No03: NOP   0;
NoXX: NOP   0;
NETWORK
TITLE =ASW_6030: Active step germinating
//      U     "MAL1S024Par".Par.FlagProcess.ProcessActive;
//      SPBN  tuen;
//
//// copy stepnr
//      L     "MAL1S024Par".Par.ParIntMachine.ActualStep;
//      T     "MAL1S024Par".Par.ParIntProcess.ActualStep;
//// set step conditions
//
//// Case where process is starting during loading
//      U     "MAL1S024Par".Par.FlagProcess.ProcessActive;
//      UN    "MAL1S024Par".Par.FlagFunction_1.StepLoading; // Step loading
//      SPBN  e003;
//// lifting devices must be in highest position
//      L       WinCoS_BIW01_09PLC1BIW01_02.Ma.Par.ParPositionTopRightUnits;
////Malting Plant OAO Belsolod Ivanonvo Weissrussland
//      L     50; // 50mm offset
//      +I    ;
//      T     "MAL1S024Par".Par.MachineValue.SOLLWERT_HUBZUG1_HOEHE;
//      L       WinCoS_BIW01_09PLC1BIW01_02.Ma.Par.ParPositionTopLeftUnits;
////Malting Plant OAO Belsolod Ivanonvo Weissrussland
//      L     50; // 50mm offset
//      +I    ;
//      T     "MAL1S024Par".Par.MachineValue.SOLLWERT_HUBZUG2_HOEHE;
//      L     5;
//      T     WinCoS_BIW01_09PLC1BIW01_02.Ma.Par.ParTolPosition;
//e003: NOP   0;
//
//// reset turning cmds
//
//// save turning cmds from prev.step
//      L     "MAL1S024Par".Par.ParIntMachine.ActualStep;
//      L     "MAL1S024Par".Par.ParIntProcess.PrevStep1stTurn;
//      <>I   ;
//      SPB   sav1;
//      U     "MAL1S024Par".Par.FlagProcess2.Turning1WithSpraying;
//      =     "MAL1S024Par".Par.Switches1.StaOn08; // Turning1WithSpraying
//      U     "MAL1S024Par".Par.FlagProcess2.Turning1WithDosing;
//      =     "MAL1S024Par".Par.Switches1.StaOn09; // Turning1WithDosing
//sav1: NOP   0;
//      L     "MAL1S024Par".Par.ParIntMachine.ActualStep;
//      L     "MAL1S024Par".Par.ParIntProcess.PrevStep2ndTurn;
//      <>I   ;
//      SPB   sav2;
//      U     "MAL1S024Par".Par.FlagProcess2.Turning2WithSpraying;
//      =     "MAL1S024Par".Par.Switches1.StaOn10; // Turning2WithSpraying
//      U     "MAL1S024Par".Par.FlagProcess2.Turning2WithDosing;
//      =     "MAL1S024Par".Par.Switches1.StaOn11; // Turning2WithDosing
//sav2: NOP   0;
//
//      SET   ;
//      R     "MAL1S024Par".Par.FlagProcess2.Turning1WithoutSpraying;
//      R     "MAL1S024Par".Par.FlagProcess2.Turning1WithSpraying;
//      R     "MAL1S024Par".Par.FlagProcess2.Turning1WithDosing;
//      R     "MAL1S024Par".Par.FlagProcess2.Turning2WithoutSpraying;
//      R     "MAL1S024Par".Par.FlagProcess2.Turning2WithSpraying;
//      R     "MAL1S024Par".Par.FlagProcess2.Turning2WithDosing;
//
//// Delta Temp to switch to next step
//      L     "MAL1S024Par".StepAct.DeltaTempSwitchpointStep;
//      L     L#0;
//      >D   ;
//      =     "MAL1S024Par".Par.FlagProcess1.DeltaTempNextStep;
//// Max Temp to switch to next step
//      L     "MAL1S024Par".StepAct.MaxTempAboveFloorStep;
//      L     L#0;
//      >D   ;
//      =     "MAL1S024Par".Par.FlagProcess1.MaxTempNextStep;
//
//// position waste air see sub 6050
//
//// basic speed fan see sub 6040
//
//// air humifidication
//      L     1;
//      L     "MAL1S024Par".StepAct.AirMoisten;   // On/Off
//      ==I;  // air humifidication on
//      U     WinCoS_BIW01_09PLC1BIW01_02.Ma.StStartedFwd; //Malting Plant OAO
//Belsolod Ivanonvo Weissrussland
//      =     "MAL1S024Par".Par.FlagProcess.AirHumidificationValve1; // air
//humifidication valve 1 on
//      U(    ; // air humifidication on
//      L     "MAL1S024Par".Par.ParIntMachine.TargetSpeedGermFan; // germinating
//fan is running
//      L     40; // fanspeed > 40%
//      >I    ; // muss noch in Istwert getauscht werden JV
//      )     ; // fanspeed > 40%
//      =     "MAL1S024Par".Par.FlagProcess.AirHumidificationValve2;
//
//// air cooling
//      L     "MAL1S024Par".StepAct.Cooling;
//      L   1;  // Activate Cooling System = 1 (yes)
//      ==I;
//      =     "MAL1S024Par".Par.FlagProcess.Cooling; // request cooling
//
//      U     "MAL1S024Par".Par.FlagProcess.ProcessActive;
//      U     "MAL1S024".PCRead.Step.StReady;
//      UN    "MAL1S024Par".Par.FlagFunction_1.StepLoading;
//      SPBN  e630;
//
//// turning 1
//      UN    "MAL1S024Par".Par.FlagProcess2.StartSecondTurningRound; // Turn
//from PrevStep
//      U(;
//      L     "MAL1S024Par".StepAct.StartTurningRound_1;
//      L     0;
//      >=D;                  // negative, no turning 1
//      );
//      U(    ;
//      O(    ; // Nach Rezept
//      L     "MAL1S024Par".ActTimeStepProcess.StepTimeActHourTotal; // Steptime
//in hours overall
//      L     "MAL1S024Par".StepAct.StartTurningRound_1;
//      ==I   ;
//      UN     WinCoS_BIW01_09PLC1BIW01_02.Ma.StAdjusted; // target position
//turning reached
//      )     ;
//      O(    ; // Selbsthaltung
//      L     "MAL1S024Par".ActTimeStepProcess.StepTimeActHourTotal; // Steptime
//in hours overall
//      L     "MAL1S024Par".StepAct.StartTurningRound_1;
//      <>I   ;
//      U     "MAL1S024Par".Par.FlagProcess2.StartFirstTurningRound;
//      )     ;
//      )     ;
//      S     "MAL1S024Par".Par.FlagProcess2.Turning1WithoutSpraying;
//      S     "MAL1S024Par".Par.FlagFunction_1.TurningStart;
//// turning 1 with spraying
//      U(    ;
//      L     1;
//      L     "MAL1S024Par".StepAct.TurningWithSpraying_1;
//      ==I;    // turning 1 with spraying on
//      U(    ;
//      L     "MAL1S024Par".Par.ParIntMachine.ActualStep;
//      L     "MAL1S024Par".Par.ParIntProcess.PrevStep1stTurn;
//      ==I   ;
//      )     ;
//      )     ;
//      O(    ;
//      L     "MAL1S024Par".Par.ParIntMachine.ActualStep;
//      L     "MAL1S024Par".Par.ParIntProcess.PrevStep1stTurn;
//      <>I   ;
//      U     "MAL1S024Par".Par.Switches1.StaOn08; // Turning1WithSpraying
//      )     ;
//      U     "MAL1S024Par".Par.FlagProcess2.Turning1WithoutSpraying;
//      S     "MAL1S024Par".Par.FlagProcess2.Turning1WithSpraying;
//// turning 1 with spraying and GA3
//      U(    ;
//      L     1;
//      L     "MAL1S024Par".StepAct.TurningWithDosing_1;
//      ==I;    // turning 1 with spraying on
//      U(    ;
//      L     "MAL1S024Par".Par.ParIntMachine.ActualStep;
//      L     "MAL1S024Par".Par.ParIntProcess.PrevStep1stTurn;
//      ==I   ;
//      )     ;
//      )     ;
//      O(    ;
//      L     "MAL1S024Par".Par.ParIntMachine.ActualStep;
//      L     "MAL1S024Par".Par.ParIntProcess.PrevStep1stTurn;
//      <>I   ;
//      U     "MAL1S024Par".Par.Switches1.StaOn09; // Turning1WithDosing
//      )     ;
//      U     "MAL1S024Par".Par.FlagProcess2.Turning1WithoutSpraying;
//      S     "MAL1S024Par".Par.FlagProcess2.Turning1WithSpraying;
//      S     "MAL1S024Par".Par.FlagProcess2.Turning1WithDosing;
//
//      U     "MAL1S024Par".Par.FlagProcess2.Turning1WithoutSpraying;
//      U     "MAL1S024Par".Par.FlagFunction_1.TurningStart;
//      UN     WinCoS_BIW01_09PLC1BIW01_02.Ma.StAdjusted; // target position
//turning reached
//      FP    "MAL1S024Par".Par.FlagProcess2.StartFirstTurningFP;
//      S     "MAL1S024Par".Par.FlagProcess2.StartFirstTurningRound;
//
//      U     WinCoS_BIW01_09PLC1BIW01_02.Ma.StAdjusted; // target position
//turning reached
//      O(    ;
//      L     "MAL1S024Par".ActTimeStepProcess.StepTimeActHourTotal; // Steptime
//in hours overall
//      L     "MAL1S024Par".StepAct.StartTurningRound_1;
//      >I    ;
//      U     WinCoS_BIW01_09PLC1BIW01_02.Ma.StAdjusted; // target position
//turning reached
//      )     ;
//      U     "MAL1S024Par".Par.FlagProcess2.StartFirstTurningRound;
//      R     "MAL1S024Par".Par.FlagProcess2.StartFirstTurningRound;
//
//      U     "MAL1S024Par".Par.FlagProcess2.StartFirstTurningFP;
//      SPB   trn1;
//      L     "MAL1S024Par".Par.ParIntMachine.ActualStep;
//      T     "MAL1S024Par".Par.ParIntProcess.PrevStep1stTurn;
//trn1: NOP   0;
//
//// turning 2
//      UN    "MAL1S024Par".Par.FlagProcess2.StartFirstTurningRound; // Unsinngie
//Rezeptwerte
//      U(;
//      L     1;
//      L     "MAL1S024Par".StepAct.StartTurningRound_2;
//      ==I    ;
//      );
//      U(    ;
//      O(    ; // Nach Rezept
//      L     "MAL1S024Par".ActTimeStepProcess.StepTimeActHourTotal; // Steptime
//in hours overall
//      L     "MAL1S024Par".StepAct.StartTurningRound_2;
//      ==I   ;
//      UN     WinCoS_BIW01_09PLC1BIW01_02.Ma.StAdjusted; // target position
//turning reached
//      )     ;
//      O(    ; // Selbsthaltung
//      L     "MAL1S024Par".ActTimeStepProcess.StepTimeActHourTotal; // Steptime
//in hours overall
//      L     "MAL1S024Par".StepAct.StartTurningRound_2;
//      <>I   ;
//      U     "MAL1S024Par".Par.FlagProcess2.StartSecondTurningRound;
//      )     ;
//      )     ;
//      S     "MAL1S024Par".Par.FlagProcess2.Turning2WithoutSpraying;
//      S     "MAL1S024Par".Par.FlagFunction_1.TurningStart;
//// turning 2 with spraying
//      U(    ;
//      L     1;
//      L     "MAL1S024Par".StepAct.TurningWithSpraying_2;
//      ==I    ;
//      U(    ;
//      L     "MAL1S024Par".Par.ParIntMachine.ActualStep;
//      L     "MAL1S024Par".Par.ParIntProcess.PrevStep2ndTurn;
//      ==I   ;
//      )     ;
//      )     ;
//      O(    ;
//      L     "MAL1S024Par".Par.ParIntMachine.ActualStep;
//      L     "MAL1S024Par".Par.ParIntProcess.PrevStep2ndTurn;
//      <>I   ;
//      U     "MAL1S024Par".Par.Switches1.StaOn10; // Turning2WithSpraying
//      )     ;
//      U     "MAL1S024Par".Par.FlagProcess2.Turning2WithoutSpraying;
//      S     "MAL1S024Par".Par.FlagProcess2.Turning2WithSpraying;
//// turning 2 with spraying and GA3
//      U(    ;
//      L     1;
//      L     "MAL1S024Par".StepAct.TurningWithDosing_2;
//      ==I;    // turning 2 with spraying and GA3 on
//      U(    ;
//      L     "MAL1S024Par".Par.ParIntMachine.ActualStep;
//      L     "MAL1S024Par".Par.ParIntProcess.PrevStep2ndTurn;
//      ==I   ;
//      )     ;
//      )     ;
//      O(    ;
//      L     "MAL1S024Par".Par.ParIntMachine.ActualStep;
//      L     "MAL1S024Par".Par.ParIntProcess.PrevStep2ndTurn;
//      <>I   ;
//      U     "MAL1S024Par".Par.Switches1.StaOn11; // Turning2WithDosing
//      )     ;
//      U     "MAL1S024Par".Par.FlagProcess2.Turning2WithoutSpraying;
//      S     "MAL1S024Par".Par.FlagProcess2.Turning2WithSpraying;
//      S     "MAL1S024Par".Par.FlagProcess2.Turning2WithDosing;
//
//      U     "MAL1S024Par".Par.FlagProcess2.Turning2WithoutSpraying;
//      U     "MAL1S024Par".Par.FlagFunction_1.TurningStart;
//      UN     WinCoS_BIW01_09PLC1BIW01_02.Ma.StAdjusted; // target position
//turning reached
//      FP    "MAL1S024Par".Par.FlagProcess2.StartSecondTurningFP;
//      S     "MAL1S024Par".Par.FlagProcess2.StartSecondTurningRound;
//
//      U     WinCoS_BIW01_09PLC1BIW01_02.Ma.StAdjusted; // target position
//turning reached
//      O(    ;
//      L     "MAL1S024Par".ActTimeStepProcess.StepTimeActHourTotal; // Steptime
//in hours overall
//      L     "MAL1S024Par".StepAct.StartTurningRound_2;
//      >I    ;
//      U     WinCoS_BIW01_09PLC1BIW01_02.Ma.StAdjusted; // target position
//turning reached
//      )     ;
//      U     "MAL1S024Par".Par.FlagProcess2.StartSecondTurningRound;
//      R     "MAL1S024Par".Par.FlagProcess2.StartSecondTurningRound;
//
//      U     "MAL1S024Par".Par.FlagProcess2.StartSecondTurningFP;
//      SPB   trn2;
//      L     "MAL1S024Par".Par.ParIntMachine.ActualStep;
//      T     "MAL1S024Par".Par.ParIntProcess.PrevStep2ndTurn;
//trn2: NOP   0;
////Fix Speed for Turning
//      U     "MAL1S024Par".Par.FlagProcess2.Turning1WithoutSpraying;
//      O     "MAL1S024Par".Par.FlagProcess2.Turning1WithSpraying;
//      O     "MAL1S024Par".Par.FlagProcess2.Turning2WithoutSpraying;
//      O     "MAL1S024Par".Par.FlagProcess2.Turning2WithSpraying;
//      U    M 50.0;
//      SPBN  SpdT;
//      L     15; // 15Hz
//      T     "MAL1S024Par".Par.MachineValue.SollwertFahrantrieb;
//SpdT: NOP   0;
//
//// find turning direction
//      U     "MAL1S024Par".Par.FlagGen.TurningStarted;
//      O(    ;
//      UN    "MAL1S024Par".Par.FlagProcess2.Turning1WithoutSpraying;
//      UN    "MAL1S024Par".Par.FlagProcess2.Turning2WithoutSpraying;
//      )     ;
//      SPB   tuen;
//      L     "MAL1S024Par".Par.ParIntMachine.TargetPosTravDriTurnRigt; // 370° =
//endposition turning right
//      T     WinCoS_BIW01_09PLC1BIW01_02.Ma.InPositionTarget; // target position
//turning reached
//
//      U(    ;
//      L     WinCoS_BIW01_09PLC1BIW01_02.Ma.OutPositionAngle;
//      L     1800;
//      <I    ; // condition turning right (clockwise)
//      )     ;
//      S     "MAL1S024Par".Par.FlagFunction_1.TurningRight;
//      S     "MAL1S024Par".Par.FlagGen.TurningStarted;
//// - Correct effect of ILO Mode
//      L       WinCoS_BIW01_09PLC1BIW01_02.Ma.Par.ParPositionTopLeftUnits;
////Malting Plant OAO Belsolod Ivanonvo Weissrussland
//      T     "MAL1S024Par".Par.MachineValue.SOLLWERT_HUBZUG1_HOEHE;
//      L       WinCoS_BIW01_09PLC1BIW01_02.Ma.Par.ParPositionTopRightUnits;
////Malting Plant OAO Belsolod Ivanonvo Weissrussland
//      T     "MAL1S024Par".Par.MachineValue.SOLLWERT_HUBZUG2_HOEHE;
//      SPB   E603   ;
//      L     "MAL1S024Par".Par.ParIntMachine.TargetPosTravDriTurnLeft; // 0° =
//endposition turning left
//      T     WinCoS_BIW01_09PLC1BIW01_02.Ma.InPositionTarget; // target position
//turning reached
//
//      U(    ;
//      L     WinCoS_BIW01_09PLC1BIW01_02.Ma.OutPositionAngle;
//      L     1800;
//      >=I   ; // condition turning left (counterclockwise)
//      )     ;
//      S     "MAL1S024Par".Par.FlagFunction_1.TurningLeft;
//      S     "MAL1S024Par".Par.FlagGen.TurningStarted;
//// - Correct effect of ILO Mode
//      L       WinCoS_BIW01_09PLC1BIW01_02.Ma.Par.ParPositionTopLeftUnits;
////Malting Plant OAO Belsolod Ivanonvo Weissrussland
//      T     "MAL1S024Par".Par.MachineValue.SOLLWERT_HUBZUG1_HOEHE;
//      L       WinCoS_BIW01_09PLC1BIW01_02.Ma.Par.ParPositionTopRightUnits;
////Malting Plant OAO Belsolod Ivanonvo Weissrussland
//      T     "MAL1S024Par".Par.MachineValue.SOLLWERT_HUBZUG2_HOEHE;
//      SPB   E603   ;
//tuen: NOP   0;
//// - Case of fast speed to protect a 2nd start during same hours as finsihed
//      O(    ; // Nach Rezept
//      L     "MAL1S024Par".ActTimeStepProcess.StepTimeActHourTotal; // Steptime
//in hours overall
//      L     "MAL1S024Par".StepAct.StartTurningRound_1;
//      ==I   ;
//      U     WinCoS_BIW01_09PLC1BIW01_02.Ma.StAdjusted; // target position
//turning reached
//      U     "MAL1S024Par".Par.FlagFunction_1.TurningStart;
//      )     ;
//      O(    ; // Nach Rezept
//      L     "MAL1S024Par".ActTimeStepProcess.StepTimeActHourTotal; // Steptime
//in hours overall
//      L     "MAL1S024Par".StepAct.StartTurningRound_2;
//      ==I   ;
//      U     WinCoS_BIW01_09PLC1BIW01_02.Ma.StAdjusted; // target position
//turning reached
//      U     "MAL1S024Par".Par.FlagFunction_1.TurningStart;
//      )     ;
//      SPB   e603;
//
//// reset turning right (clockwise)
//      U     "MAL1S024Par".Par.FlagFunction_1.TurningRight;
//      U(    ;
//      O      WinCoS_BIW01_09PLC1BIW01_02.Ma.StAdjusted; // target position
//turning reached
//      O(    ;
//      L     WinCoS_BIW01_09PLC1BIW01_02.Ma.OutPositionAngle;
//      L     WinCoS_BIW01_09PLC1BIW01_02.Ma.Par.ParTolPosition;
//      +I    ;
//      L     "MAL1S024Par".Par.ParIntMachine.TargetPosTravDriTurnRigt;
//      >=I   ;
//      )     ;
//      )     ;
//      R     "MAL1S024Par".Par.FlagFunction_1.TurningRight;
//      R     "MAL1S024Par".Par.FlagFunction_1.TurningStart;
//
//// reset turning left (counterclockwise)
//      U     "MAL1S024Par".Par.FlagFunction_1.TurningLeft;
//      U(    ;
//      O     WinCoS_BIW01_09PLC1BIW01_02.Ma.StAdjusted; // target position
//turning reached
//      O(    ;
//      L     WinCoS_BIW01_09PLC1BIW01_02.Ma.OutPositionAngle;
//      L     WinCoS_BIW01_09PLC1BIW01_02.Ma.Par.ParTolPosition;
//      -I    ;
//      L     "MAL1S024Par".Par.ParIntMachine.TargetPosTravDriTurnLeft;
//      <=I   ;
//      )     ;
//      )     ;
//      R     "MAL1S024Par".Par.FlagFunction_1.TurningLeft;
//      R     "MAL1S024Par".Par.FlagFunction_1.TurningStart;
//
//// reset turning flag
//      U     "MAL1S024Par".Par.FlagGen.TurningStarted;
//      UN    "MAL1S024Par".Par.FlagProcess2.Turning1WithoutSpraying;
//      UN    "MAL1S024Par".Par.FlagProcess2.Turning2WithoutSpraying;
//      O(    ;
//      U     "MAL1S024Par".Par.FlagGen.TurningStarted;
//      U     WinCoS_BIW01_09PLC1BIW01_02.Ma.StAdjusted; // target position
//turning reached
//      )     ;
//      ON    "MAL1S024Par".Par.FlagProcess.ProcessActive;
//      R     "MAL1S024Par".Par.FlagGen.TurningStarted;
//      R     "MAL1S024Par".Par.FlagProcess2.Turning1WithoutSpraying;
//      R     "MAL1S024Par".Par.FlagProcess2.Turning2WithoutSpraying;
//      R     "MAL1S024Par".Par.FlagFunction_1.TurningStart;
//e630: NOP   0;
//      UN    "MAL1S024Par".Par.FlagProcess.ProcessActive;
//      R     "MAL1S024Par".Par.FlagProcess2.StartFirstTurningRound;
//      R     "MAL1S024Par".Par.FlagProcess2.StartSecondTurningRound;
//
//e603: NOP   0;
//E603: NOP   0;
      U     "MAL1S024Par".Par.FlagProcess.ProcessActive;
      SPBN  tuen;

// copy stepnr
      L     "MAL1S024Par".Par.ParIntMachine.ActualStep;
      T     "MAL1S024Par".Par.ParIntProcess.ActualStep;
// set step conditions

// reset turning cmds

// save turning cmds from prev.step
      L     "MAL1S024Par".Par.ParIntMachine.ActualStep;
      L     "MAL1S024Par".Par.ParIntProcess.PrevStep1stTurn;
      <>I   ;
      SPB   sav1;
      U     "MAL1S024Par".Par.FlagProcess2.Turning1WithSpraying;
      =     "MAL1S024Par".Par.Switches1.StaOn08; // Turning1WithSpraying
      U     "MAL1S024Par".Par.FlagProcess2.Turning1WithDosing;
      =     "MAL1S024Par".Par.Switches1.StaOn09; // Turning1WithDosing
sav1: NOP   0;
      L     "MAL1S024Par".Par.ParIntMachine.ActualStep;
      L     "MAL1S024Par".Par.ParIntProcess.PrevStep2ndTurn;
      <>I   ;
      SPB   sav2;
      U     "MAL1S024Par".Par.FlagProcess2.Turning2WithSpraying;
      =     "MAL1S024Par".Par.Switches1.StaOn10; // Turning2WithSpraying
      U     "MAL1S024Par".Par.FlagProcess2.Turning2WithDosing;
      =     "MAL1S024Par".Par.Switches1.StaOn11; // Turning2WithDosing
sav2: NOP   0;

      SET   ;
      R     "MAL1S024Par".Par.FlagProcess2.Turning1WithoutSpraying;
      R     "MAL1S024Par".Par.FlagProcess2.Turning1WithSpraying;
      R     "MAL1S024Par".Par.FlagProcess2.Turning1WithDosing;
      R     "MAL1S024Par".Par.FlagProcess2.Turning2WithoutSpraying;
      R     "MAL1S024Par".Par.FlagProcess2.Turning2WithSpraying;
      R     "MAL1S024Par".Par.FlagProcess2.Turning2WithDosing;

// Delta Temp to switch to next step
      L     "MAL1S024Par".StepAct.DeltaTempSwitchpointStep;
      L     L#0;
      >D    ;
      =     "MAL1S024Par".Par.FlagProcess1.DeltaTempNextStep;
// Max Temp to switch to next step
      L     "MAL1S024Par".StepAct.MaxTempAboveFloorStep;
      L     L#0;
      >D    ;
      =     "MAL1S024Par".Par.FlagProcess1.MaxTempNextStep;

// position waste air see sub 6050

// basic speed fan see sub 6040

// air humifidication

// air cooling
      L     "MAL1S024Par".StepAct.Cooling;
      L     1; // Activate Cooling System = 1 (yes)
      ==I   ;
      =     "MAL1S024Par".Par.FlagProcess.Cooling; // request cooling

      U     "MAL1S024Par".Par.FlagProcess.ProcessActive;
      U     "MAL1S024".PCRead.Step.StReady;
      UN    "MAL1S024Par".Par.FlagFunction_1.StepLoading;
      SPBN  e630;

// turning 1
      UN    "MAL1S024Par".Par.FlagProcess2.StartSecondTurningRound; // Turn from PrevStep
      U(    ;
      L     "MAL1S024Par".StepAct.StartTurningRound_1;
      L     0;
      >=I   ; // negative, no turning 1
      )     ;
      U(    ;
      O(    ; // Nach Rezept
      L     "MAL1S024Par".ActTimeStepProcess.StepTimeActHourTotal; // Steptime in hours overall
      L     "MAL1S024Par".StepAct.StartTurningRound_1;
      ==I   ;
      UN    "G245M".A_2811_MXZ41MA.Ma.StAdjusted; // target position turning reached
      )     ;
      O(    ; // Selbsthaltung
      L     "MAL1S024Par".ActTimeStepProcess.StepTimeActHourTotal; // Steptime in hours overall
      L     "MAL1S024Par".StepAct.StartTurningRound_1;
      <>I   ;
      U     "MAL1S024Par".Par.FlagProcess2.StartFirstTurningRound;
      )     ;
      )     ;
      S     "MAL1S024Par".Par.FlagProcess2.Turning1WithoutSpraying;
      S     "MAL1S024Par".Par.FlagFunction_1.TurningStart;
// turning 1 with spraying
      U(    ;
      L     1;
      L     "MAL1S024Par".StepAct.TurningWithSpraying_1;
      ==I   ; // turning 1 with spraying on
      U(    ;
      L     "MAL1S024Par".Par.ParIntMachine.ActualStep;
      L     "MAL1S024Par".Par.ParIntProcess.PrevStep1stTurn;
      ==I   ;
      )     ;
      )     ;
      O(    ;
      L     "MAL1S024Par".Par.ParIntMachine.ActualStep;
      L     "MAL1S024Par".Par.ParIntProcess.PrevStep1stTurn;
      <>I   ;
      U     "MAL1S024Par".Par.Switches1.StaOn08; // Turning1WithSpraying
      )     ;
      U     "MAL1S024Par".Par.FlagProcess2.Turning1WithoutSpraying;
      S     "MAL1S024Par".Par.FlagProcess2.Turning1WithSpraying;
// turning 1 with spraying and GA3
      U(    ;
      L     1;
      L     "MAL1S024Par".StepAct.TurningWithDosing_1;
      ==I   ; // turning 1 with spraying on
      U(    ;
      L     "MAL1S024Par".Par.ParIntMachine.ActualStep;
      L     "MAL1S024Par".Par.ParIntProcess.PrevStep1stTurn;
      ==I   ;
      )     ;
      )     ;
      O(    ;
      L     "MAL1S024Par".Par.ParIntMachine.ActualStep;
      L     "MAL1S024Par".Par.ParIntProcess.PrevStep1stTurn;
      <>I   ;
      U     "MAL1S024Par".Par.Switches1.StaOn09; // Turning1WithDosing
      )     ;
      U     "MAL1S024Par".Par.FlagProcess2.Turning1WithoutSpraying;
      S     "MAL1S024Par".Par.FlagProcess2.Turning1WithSpraying;
      S     "MAL1S024Par".Par.FlagProcess2.Turning1WithDosing;

//BRT070410 - wird einen Zyklus später gesetzt
      U     "MAL1S024Par".Par.FlagProcess2.StartFirstDosingFP;
      S     "MAL1S024Par".Par.FlagProcess2.StartFirstTurningRound;

      U     "MAL1S024Par".Par.FlagProcess2.Turning1WithoutSpraying;
      U     "MAL1S024Par".Par.FlagFunction_1.TurningStart;
//BRT060310      UN    "G245M".A_2811_MXZ41MA.Ma.StAdjusted    // target position turning reached
      UN    "G245M".A_2811_MXZ41MA.Ma.OutAdjusted; // target position turning reached
      FP    "MAL1S024Par".Par.FlagProcess2.StartFirstTurningFP;
      =     "MAL1S024Par".Par.FlagProcess2.StartFirstDosingFP;
//BRT070410      S     "MAL1S024Par".Par.FlagProcess2.StartFirstTurningRound

      U     "MAL1S024Par".Par.FlagProcess2.StartFirstDosingFP;
      U     "MAL1S024Par".Par.FlagProcess2.StartFirstTurningFP;
      SPBN  trn1;
      L     "MAL1S024Par".Par.ParIntMachine.ActualStep;
      T     "MAL1S024Par".Par.ParIntProcess.PrevStep1stTurn;
trn1: NOP   0;

//BRT060310      U     "G245M".A_2811_MXZ41MA.Ma.StAdjusted    // target position turning reached
      U     "G245M".A_2811_MXZ41MA.Ma.OutAdjusted; // target position turning reached
      O(    ;
      L     "MAL1S024Par".ActTimeStepProcess.StepTimeActHourTotal; // Steptime in hours overall
      L     "MAL1S024Par".StepAct.StartTurningRound_1;
      >I    ;
      U(    ;
      O     "G245M".A_2811_MXZ41MA.Ma.OutAdjusted; // target position turning reached
      O(    ;
//BRT070310      UN    "G245M".A_2811_BZS46.StTrue // stop fan side
//BRT070310      U     "G245M".A_2811_BZS44.StTrue // stop discharge side
      U     "G245M".A_2811_BZS46.StTrue; // stop end side
      UN    "G245M".A_2811_BZS44.StTrue; // stop zeroposition
      U     "MAL1S024Par".Par.FlagFunction_1.TurningRight;
      )     ;
      O(    ;
//BRT070310      U     "G245M".A_2811_BZS46.StTrue // stop fan side
//BRT070310      UN    "G245M".A_2811_BZS44.StTrue // stop discharge side
      UN    "G245M".A_2811_BZS46.StTrue; // stop end side
      U     "G245M".A_2811_BZS44.StTrue; // stop zeroposition
      U     "MAL1S024Par".Par.FlagFunction_1.TurningLeft;
      )     ;
      )     ;
      )     ;
      O(    ;
      L     "MAL1S024Par".StepAct.StartTurningRound_1;
//BRT070310      L     0
//BRT070310      <D                                // negative, no turning 1
      L     -1; //BRT070310
      ==I   ; //BRT070310
      )     ;
      U     "MAL1S024Par".Par.FlagProcess2.StartFirstTurningRound;
      R     "MAL1S024Par".Par.FlagProcess2.StartFirstTurningRound;
      R     "MAL1S024Par".Par.Switches1.StaOn08; // Turning1WithSpraying
      R     "MAL1S024Par".Par.Switches1.StaOn09; // Turning1WithDosing

// turning 2
      UN    "MAL1S024Par".Par.FlagProcess2.StartFirstTurningRound; // Unsinnige Rezeptwerte
      U(    ;
//      L     1
      L     "MAL1S024Par".StepAct.StartTurningRound_2;
//      <>I
      L     0;
      >=I   ;
      )     ;
      U(    ;
      O(    ; // Nach Rezept
      L     "MAL1S024Par".ActTimeStepProcess.StepTimeActHourTotal; // Steptime in hours overall
      L     "MAL1S024Par".StepAct.StartTurningRound_2;
      ==I   ;
      UN    "G245M".A_2811_MXZ41MA.Ma.StAdjusted; // target position turning reached
      )     ;
      O(    ; // Selbsthaltung
      L     "MAL1S024Par".ActTimeStepProcess.StepTimeActHourTotal; // Steptime in hours overall
      L     "MAL1S024Par".StepAct.StartTurningRound_2;
      <>I   ;
      U     "MAL1S024Par".Par.FlagProcess2.StartSecondTurningRound;
      )     ;
      )     ;
      S     "MAL1S024Par".Par.FlagProcess2.Turning2WithoutSpraying;
      S     "MAL1S024Par".Par.FlagFunction_1.TurningStart;
// turning 2 with spraying
      U(    ;
      L     1;
      L     "MAL1S024Par".StepAct.TurningWithSpraying_2;
      ==I   ;
      U(    ;
      L     "MAL1S024Par".Par.ParIntMachine.ActualStep;
      L     "MAL1S024Par".Par.ParIntProcess.PrevStep2ndTurn;
      ==I   ;
      )     ;
      )     ;
      O(    ;
      L     "MAL1S024Par".Par.ParIntMachine.ActualStep;
      L     "MAL1S024Par".Par.ParIntProcess.PrevStep2ndTurn;
      <>I   ;
      U     "MAL1S024Par".Par.Switches1.StaOn10; // Turning2WithSpraying
      )     ;
      U     "MAL1S024Par".Par.FlagProcess2.Turning2WithoutSpraying;
      S     "MAL1S024Par".Par.FlagProcess2.Turning2WithSpraying;
// turning 2 with spraying and GA3
      U(    ;
      L     1;
      L     "MAL1S024Par".StepAct.TurningWithDosing_2;
      ==I   ; // turning 2 with spraying and GA3 on
      U(    ;
      L     "MAL1S024Par".Par.ParIntMachine.ActualStep;
      L     "MAL1S024Par".Par.ParIntProcess.PrevStep2ndTurn;
      ==I   ;
      )     ;
      )     ;
      O(    ;
      L     "MAL1S024Par".Par.ParIntMachine.ActualStep;
      L     "MAL1S024Par".Par.ParIntProcess.PrevStep2ndTurn;
      <>I   ;
      U     "MAL1S024Par".Par.Switches1.StaOn11; // Turning2WithDosing
      )     ;
      U     "MAL1S024Par".Par.FlagProcess2.Turning2WithoutSpraying;
      S     "MAL1S024Par".Par.FlagProcess2.Turning2WithSpraying;
      S     "MAL1S024Par".Par.FlagProcess2.Turning2WithDosing;

//BRT070410 - wird einen Zyklus später gesetzt
      U     "MAL1S024Par".Par.FlagProcess2.StartSecondDosingFP;
      S     "MAL1S024Par".Par.FlagProcess2.StartSecondTurningRound;

      U     "MAL1S024Par".Par.FlagProcess2.Turning2WithoutSpraying;
      U     "MAL1S024Par".Par.FlagFunction_1.TurningStart;
//BRT060310      UN    "G245M".A_2811_MXZ41MA.Ma.StAdjusted    // target position turning reached
      UN    "G245M".A_2811_MXZ41MA.Ma.OutAdjusted; // target position turning reached
      FP    "MAL1S024Par".Par.FlagProcess2.StartSecondTurningFP;
      =     "MAL1S024Par".Par.FlagProcess2.StartSecondDosingFP;
//BRT070410      S     "MAL1S024Par".Par.FlagProcess2.StartSecondTurningRound

      U     "MAL1S024Par".Par.FlagProcess2.StartSecondDosingFP;
      U     "MAL1S024Par".Par.FlagProcess2.StartSecondTurningFP;
      SPBN  trn2;
      L     "MAL1S024Par".Par.ParIntMachine.ActualStep;
      T     "MAL1S024Par".Par.ParIntProcess.PrevStep2ndTurn;
trn2: NOP   0;

//BRT060310      U    "G245M".A_2811_MXZ41MA.Ma.StAdjusted    // target position turning reached
      U     "G245M".A_2811_MXZ41MA.Ma.OutAdjusted; // target position turning reached
      O(    ;
      L     "MAL1S024Par".ActTimeStepProcess.StepTimeActHourTotal; // Steptime in hours overall
      L     "MAL1S024Par".StepAct.StartTurningRound_2;
      >I    ;
      U(    ;
      O     "G245M".A_2811_MXZ41MA.Ma.OutAdjusted; // target position turning reached
      O(    ;
      UN    "G245M".A_2811_BZS46.StTrue; // stop fan side
      U     "G245M".A_2811_BZS44.StTrue; // stop discharge side
      U     "MAL1S024Par".Par.FlagFunction_1.TurningRight;
      )     ;
      O(    ;
      U     "G245M".A_2811_BZS46.StTrue; // stop fan side
      UN    "G245M".A_2811_BZS44.StTrue; // stop discharge side
      U     "MAL1S024Par".Par.FlagFunction_1.TurningLeft;
      )     ;
      )     ;
      )     ;
      O(    ;
      L     "MAL1S024Par".StepAct.StartTurningRound_2;
//BRT070310      L     0
//BRT070310      <D                                // negative, no turning 2
      L     -1; //BRT070310
      ==I   ; //BRT070310
      )     ;
      U     "MAL1S024Par".Par.FlagProcess2.StartSecondTurningRound;
      R     "MAL1S024Par".Par.FlagProcess2.StartSecondTurningRound;
      R     "MAL1S024Par".Par.Switches1.StaOn10; // Turning2WithSpraying
      R     "MAL1S024Par".Par.Switches1.StaOn11; // Turning2WithDosing

      L     3600;
      T     "MAL1S024Par".Par.ParIntMachine.TargetPosTravDriTurnRigt; // 360° = endposition turning right

// find turning direction spez. APU: right ==> forward, left ==> reverse
      U     "MAL1S024Par".Par.FlagGen.TurningStarted;
      O(    ;
      UN    "MAL1S024Par".Par.FlagProcess2.Turning1WithoutSpraying;
      UN    "MAL1S024Par".Par.FlagProcess2.Turning2WithoutSpraying;
      )     ;
      SPB   tuen;
      L     "MAL1S024Par".Par.ParIntMachine.TargetPosTravDriTurnRigt; // 360° = endposition turning right
      T     "G245M".A_2811_MXZ41MA.Ma.InPositionTarget; // target position turning

      U(    ;
      L     "G245M".A_2811_MXZ41MA.Ma.OutPositionAngle;
      L     1800;
      <I    ; // condition turning right (clockwise)
      )     ;
//BRT070310      O     "G245M".A_2811_BZS46.StTrue // stop end side
//BRT070310      UN    "G245M".A_2811_BZS44.StTrue // stop zeroposition
      O     "G245M".A_2811_BZS44.StTrue; // stop zeroposition  //BRT070310
      UN    "G245M".A_2811_BZS46.StTrue; //stop end side   //BRT070310
      S     "MAL1S024Par".Par.FlagFunction_1.TurningRight;
      S     "MAL1S024Par".Par.FlagGen.TurningStarted;
      SPB   E603;
      L     "MAL1S024Par".Par.ParIntMachine.TargetPosTravDriTurnLeft; // 0° = endposition turning left
      T     "G245M".A_2811_MXZ41MA.Ma.InPositionTarget; // target position turning

      U(    ;
      L     "G245M".A_2811_MXZ41MA.Ma.OutPositionAngle;
      L     1800;
      >=I   ; // condition turning left (counterclockwise)
      )     ;
//BRT070310      O     "G245M".A_2811_BZS44.StTrue // stop end side
//BRT070310      UN    "G245M".A_2811_BZS46.StTrue // stop zeroposition
      O     "G245M".A_2811_BZS46.StTrue; // stop zeroposition  //BRT070310
      UN    "G245M".A_2811_BZS44.StTrue; //stop end side   //BRT070310
      S     "MAL1S024Par".Par.FlagFunction_1.TurningLeft;
      S     "MAL1S024Par".Par.FlagGen.TurningStarted;
      SPB   E603;
tuen: NOP   0;

// reset turning right (clockwise)
      U     "MAL1S024Par".Par.FlagFunction_1.TurningRight;
      U(    ;
//      O     "G242M"._2111_MXZ41MA.Ma.StAdjusted    // target position turning reached
      O(    ;
      L     "G245M".A_2811_MXZ41MA.Ma.OutPositionAngle;
      L     "G245M".A_2811_MXZ41MA.Ma.Par.ParTolPosition;
      +I    ;
      L     "MAL1S024Par".Par.ParIntMachine.TargetPosTravDriTurnRigt;
      >=I   ;
      )     ;
//BRT070310      O     "G245M".A_2811_BZS44.StTrue // stop end side
      O     "G245M".A_2811_BZS46.StTrue; // stop zeroposition
      )     ;
      R     "MAL1S024Par".Par.FlagFunction_1.TurningRight;
      R     "MAL1S024Par".Par.FlagFunction_1.TurningStart;

// reset turning left (counterclockwise)
      U     "MAL1S024Par".Par.FlagFunction_1.TurningLeft;
      U(    ;
//      O     "G242M"._2111_MXZ41MA.Ma.StAdjusted    // target position turning reached
      O(    ;
      L     "G245M".A_2811_MXZ41MA.Ma.OutPositionAngle;
      L     "G245M".A_2811_MXZ41MA.Ma.Par.ParTolPosition;
      -I    ;
      L     "MAL1S024Par".Par.ParIntMachine.TargetPosTravDriTurnLeft;
      <=I   ;
      )     ;
      O     "G245M".A_2811_BZS44.StTrue; // stop end side
//BRT070310      O     "G245M".A_2811_BZS46.StTrue // stop zeroposition
      )     ;
      R     "MAL1S024Par".Par.FlagFunction_1.TurningLeft;
      R     "MAL1S024Par".Par.FlagFunction_1.TurningStart;

// - Case of fast speed to protect a 2nd start during same hours as finsihed
      U     "MAL1S024Par".Par.FlagGen.TurningStarted;
//====>BRT070310      UN    "MAL1S024Par".Par.FlagProcess.ProcessEnd    // JV210808 to finish last turning
      U(    ;
      U     "MAL1S024Par".Par.FlagProcess2.Turning1WithoutSpraying;
      O     "MAL1S024Par".Par.FlagProcess2.Turning2WithoutSpraying;
      UN    "MAL1S024Par".Par.FlagProcess.ProcessEnd; // JV210808 to finish last turning
      )     ;
      UN    "MAL1S024StepValues".StartStep; // start step for average calculating
      U(    ;
      O(    ; // Nach Rezept
      U(    ;
      L     "MAL1S024Par".ActTimeStepProcess.StepTimeActHourTotal; // Steptime in hours overall
      L     "MAL1S024Par".StepAct.StartTurningRound_1;
      ==I   ; // JV 250808
      )     ;
//      UN    "MAL1S024Par".Par.FlagProcess2.StartFirstTurningRound    // JV 250808
      U     "G245M".A_2811_MXZ41MA.Ma.OutAdjusted; // target position turning reached
      )     ;
      O(    ; // Nach Rezept
      U(    ;
      L     "MAL1S024Par".ActTimeStepProcess.StepTimeActHourTotal; // Steptime in hours overall
      L     "MAL1S024Par".StepAct.StartTurningRound_2;
      ==I   ; // JV 250808
      )     ;
//      UN    "MAL1S024Par".Par.FlagProcess2.StartSecondTurningRound    // JV 250808
      U     "G245M".A_2811_MXZ41MA.Ma.OutAdjusted; // target position turning reached
//<====BRT070310
      )     ;
      )     ;
      O(    ;
      UN    "G245M".A_2811_MXZ41MA.Ma.OutAdjusted; // target position turning reached
      UN    "MAL1S024Par".Par.FlagFunction_1.StepUnloading;
      )     ;
      SPB   e603;

// reset turning flag
      U     "MAL1S024Par".Par.FlagGen.TurningStarted;
      ON    "MAL1S024Par".Par.FlagProcess.ProcessActive;
      R     "MAL1S024Par".Par.FlagGen.TurningStarted;
      R     "MAL1S024Par".Par.FlagProcess2.Turning1WithoutSpraying;
      R     "MAL1S024Par".Par.FlagProcess2.Turning2WithoutSpraying;
      R     "MAL1S024Par".Par.FlagProcess2.Turning1WithSpraying;
      R     "MAL1S024Par".Par.FlagProcess2.Turning2WithSpraying;
      R     "MAL1S024Par".Par.FlagProcess2.Turning1WithDosing;
      R     "MAL1S024Par".Par.FlagProcess2.Turning2WithDosing;
      R     "MAL1S024Par".Par.FlagFunction_1.TurningStart;
      R     "MAL1S024Par".Par.FlagProcess2.StartFirstTurningRound; // JV 250808
      R     "MAL1S024Par".Par.FlagProcess2.StartSecondTurningRound; // JV 250808
      SET   ;
      R     "MAL1S024StepValues".StartStep; // start step for average calculating
e630: NOP   0;
      UN    "MAL1S024Par".Par.FlagProcess.ProcessActive;
      R     "MAL1S024Par".Par.FlagProcess2.StartFirstTurningRound;
      R     "MAL1S024Par".Par.FlagProcess2.StartSecondTurningRound;
      R     "MAL1S024Par".Par.Switches1.StaOn08; // Turning1WithSpraying
      R     "MAL1S024Par".Par.Switches1.StaOn09; // Turning1WithDosing
      R     "MAL1S024Par".Par.Switches1.StaOn10; // Turning2WithSpraying
      R     "MAL1S024Par".Par.Switches1.StaOn11; // Turning2WithDosing

      L     "G245M".A_2811_MXZ41MA.Ma.OutPositionAngle;
      T     "G245M".A_2811_MXZ41MA.Ma.OutPositionAngle;

      L     "G245M".A_2811_MXZ41MA.Ma.OutPositionRel;
      T     "G245M".A_2811_MXZ41MA.Ma.OutPositionRel;

e603: NOP   0;
E603: NOP   0;

NETWORK
TITLE =ASW_6040: Set fanspeed by delta-t
//Die Drehzahl des Ventilators wird zwischen dem Rezeptsollwert, als Untere
//Grenze, und 100% oder Rezeptsollwert, als obere Grenze, geregelt. Die Regelung
//erfolgt nach folgendem Prinzip:
//"Delta-T" ist die Differenz zwischen der Soll-Temperatur (Rezeptsollwert) unter
//der Horde und der gemessenen Ist-Temperatur über der Horde.
//Steigt die Ist-Temperatur über der Horde und "Delta-T" wird > als der Sollwert
//im Rezept, so wird die Drehzahl des Ventilators stufenweise erhöht. Maximale
//Drehzahl ist 100% oder Rezeptsollwert.
//Sinkt die Ist-Temperatur über der Horde und "Delta-T" wird < als der Sollwert
//im
//Rezept, so wird die Drehzahl des Ventilators stufenweise verringert. Minimale
//Drehzahl ist der Rezeptsollwert.
//Die Rampen (Stufen) werden durch den Technologen festgelegt und in Programmcode
//eingetragen. Es sind keine Rezeptsollwerte.
      NOP   0;
//====>BRT070310
// recipe setpoint
//      L     "MAL1S024Par".StepAct.SpeedVentilatorBasic
//      L     0
//      ==I                               // no fan during turning
//      SPB   e604                        // JV040908
      UN(   ;
      U(    ;
      L     "MAL1S024Par".Par.ParIntMachine.ActualStep;
      L     1;
      ==I   ;
      )     ;
      UN(   ;
      L     "MAL1S024Par".Par.ProcessValue.StepTimeAct; // in ms
      L     L#1000; // in first secunde steptime
      >D    ;
      )     ;
      )     ;
// BRT070310 - berechneter Targetwert darf nur bei StepNr.1 oder! Rezeptwert-Änderung überschrieben werden
      U(    ;
      L     "MAL1S024Par".StepAct.SpeedVentilatorBasic;
      L     "MAL1S024Par".Par.ParIntProcess.Value23; // Rezeptwert vor Änderung
      ==D   ;
      )     ;
      SPB   regu;
      L     "MAL1S024Par".StepAct.SpeedVentilatorBasic;
      T     "MAL1S024Par".Par.ParIntProcess.Value23; // Rezeptwert vor Änderung
      SPA   Summ;
regu: NOP   0;

// BRT070310 - nicht nötig, da obige Änderung bei Änderung Rezeptwert (Modify) auch Target-Wert neu lädt
//      U     "MAL1S024".ToASW.CmdModify
//      SPB   Summ
//<====BRT070310

// Setpoint
      L     "MAL1S024Par".StepAct.TemperaturAboveFloor;
      L     "MAL1S024Par".StepAct.TemperaturBelowFloor;
      -D    ;
      T     "MAL1S024Par".Par.ProcessValue.SetpointDeltaTempDint;
// actual value
      L     "G248M".A_2891_BTE02.OutValueUnits; //AIR TEMPERATURE ABOVE FLOOR
      L     "G248M".A_2891_BTE01.OutValueUnits; //AIR TEMPERATURE BELOW FLOOR
      -D    ;
      L     L#10; //BRT070310
      /D    ; //BRT070310
      T     "MAL1S024Par".Par.ProcessValue.ActValueDeltaTempDint;
// flags to inc/dec
      L     "MAL1S024Par".Par.ProcessValue.SetpointDeltaTempDint;
      -D    ;
      T     "MAL1S024Par".Par.ProcessValue.ResultDeltaTemp;
      L     L#0;
      >D    ;
      =     "MAL1S024Par".Par.FlagProcess1.DeltaTempPlus;
      <D    ;
      =     "MAL1S024Par".Par.FlagProcess1.DeltaTempMinus;

      U     "MAL1S024Par".Par.FlagProcess1.DeltaTempPlus;
//BRT200310      U     "SYS_Scan0_Tick1min"
      U     "SYS_Scan0_Tick30s"; //Scan0_Tick30s
      SPBN  dec;
      L     "MAL1S024Par".Par.ParIntMachine.TargetSpeedGermFan;
      L     100; // linmit max
      >=I   ;
      O(    ; //JV160710 =====>
      TAK   ;
      L     "MAL1S024Par".StepAct.SpeedVentilatorMaximal;
      >=I   ;
      U(    ;
      L     "MAL1S024Par".StepAct.SpeedVentilatorMaximal;
      L     "MAL1S024Par".StepAct.SpeedVentilatorBasic;
      >=I   ;
      )     ;
      )     ; //JV160710 <=====
      SPB   dec;
      L     "MAL1S024Par".Par.ParIntMachine.TargetSpeedGermFan;
      L     1;
      +I    ;
      T     "MAL1S024Par".Par.ParIntMachine.TargetSpeedGermFan;
      SPA   e604;
dec:  NOP   0;
      U     "MAL1S024Par".Par.FlagProcess1.DeltaTempMinus;
      O(    ; //JV160710 =====>
      L     "MAL1S024Par".Par.ParIntMachine.TargetSpeedGermFan;
      L     "MAL1S024Par".StepAct.SpeedVentilatorMaximal;
      >I    ;
      )     ; //JV160710 <=====
//BRT200310      U     "SYS_Scan0_Tick1min"
      U     "SYS_Scan0_Tick30s"; //Scan0_Tick30s
      SPBN  e604;
      L     "MAL1S024Par".Par.ParIntMachine.TargetSpeedGermFan;
      L     "MAL1S024Par".StepAct.SpeedVentilatorBasic; // linmit min
      <=I   ;
      SPB   e604;
      L     "MAL1S024Par".Par.ParIntMachine.TargetSpeedGermFan;
      L     1;
      -I    ;
      T     "MAL1S024Par".Par.ParIntMachine.TargetSpeedGermFan;
      SPA   e604;

Summ: NOP   0;
      L     "MAL1S024Par".StepAct.SpeedVentilatorBasic;
      T     "MAL1S024Par".Par.ParIntMachine.TargetSpeedGermFan;
      U     "MAL1S024Par".Par.FlagProcess.ProcessEnd; // JV030908
      UN    "MAL1S024".PCRead.Step.StEmptying;
      UN    "MAL1S024".PCRead.Step.StEmptied;
      SPBN  e604;
      L     "MAL1S024Par".Par.ParIntProcess.SavedTargetSpeedGermFan;
      T     "MAL1S024Par".Par.ParIntMachine.TargetSpeedGermFan;
e604: NOP   0;
// store actual setpoint
      U     "MAL1S024Par".Par.FlagProcess.ProcessActive;
      U(    ;
      L     "MAL1S024Par".StepAct.SpeedVentilatorBasic;
      L     0; // setpoint recipe > 0
      >I    ;
      )     ;
      SPBN  E604;
      L     "MAL1S024Par".StepAct.SpeedVentilatorBasic;
      T     "MAL1S024Par".Par.ParIntProcess.SavedTargetSpeedGermFan;
E604: NOP   0;
//-------------------------------------------------------------------------------------------------
//--- Ventilator 2 einzeln geregelt ---
      UN(   ;
      U(    ;
      L     "MAL1S024Par".Par.ParIntMachine.ActualStep;
      L     1;
      ==I   ;
      )     ;
      UN(   ;
      L     "MAL1S024Par".Par.ProcessValue.StepTimeAct; // in ms
      L     L#1000; // in first secunde steptime
      >D    ;
      )     ;
      )     ;
// BRT040310 - berechneter Targetwert darf nur bei StepNr.1 oder! Rezeptwert-Änderung überschrieben werden
      U(    ;
      L     "MAL1S024Par".StepAct.SpeedVentilatorBasic;
      L     "MAL1S024Par".Par.ParIntProcess.Value25; // Rezeptwert vor Änderung
      ==D   ;
      )     ;
      SPB   reg1;
      L     "MAL1S024Par".StepAct.SpeedVentilatorBasic;
      T     "MAL1S024Par".Par.ParIntProcess.Value25; // Rezeptwert vor Änderung
      SPA   Sum1;
reg1: NOP   0;
// Setpoint
      L     "MAL1S024Par".StepAct.TemperaturAboveFloor;
      L     "MAL1S024Par".StepAct.TemperaturBelowFloor;
      -D    ;
      T     "MAL1S024Par".Par.ProcessValue.Value13; // Setpoint Delta Temp
// actual value
      L     "G248M".A_2891_BTE04.OutValueUnits; //AIR TEMPERATURE ABOVE FLOOR
      L     "G248M".A_2891_BTE03.OutValueUnits; //AIR TEMPERATURE BELOW FLOOR
      -D    ;
      L     L#10; //BRT060310
      /D    ; //BRT060310
      T     "MAL1S024Par".Par.ProcessValue.Value14; // Actual Value Delta Temp
// flags to inc/dec
      L     "MAL1S024Par".Par.ProcessValue.Value13; // Setpoint Delta Temp
      -D    ;
      T     "MAL1S024Par".Par.ProcessValue.Value15; // Result Delta Temp
      L     L#0;
      >D    ;
      =     "MAL1S024Par".Par.FlagProcess1.Inf23; // Delta Temp Plus
      <D    ;
      =     "MAL1S024Par".Par.FlagProcess1.Inf24; // Delta Temp Minus

      U     "MAL1S024Par".Par.FlagProcess1.Inf23; // Delta Temp Plus
//BRT203010      U     "SYS_Scan0_Tick1min"
      U     "SYS_Scan0_Tick30s"; //Scan0_Tick30s
      SPBN  dec1;
      L     "MAL1S024Par".Par.ParIntProcess.Value26; // Target Speed GermFan 2
      L     100; // linmit max
      >=I   ;
      O(    ; //JV160710 =====>
      TAK   ;
      L     "MAL1S024Par".StepAct.SpeedVentilatorMaximal;
      >=I   ;
      U(    ;
      L     "MAL1S024Par".StepAct.SpeedVentilatorMaximal;
      L     "MAL1S024Par".StepAct.SpeedVentilatorBasic;
      >=I   ;
      )     ;
      )     ; //JV160710 <=====
      SPB   dec1;
      L     "MAL1S024Par".Par.ParIntProcess.Value26; // Target Speed GermFan 2
      L     1;
      +I    ;
      T     "MAL1S024Par".Par.ParIntProcess.Value26; // Target Speed GermFan 2
      SPA   e614;
dec1: NOP   0;
      U     "MAL1S024Par".Par.FlagProcess1.Inf24; // Delta Temp Minus
      O(    ; //JV160710 =====>
      L     "MAL1S024Par".Par.ParIntProcess.Value26; // Target Speed GermFan 2
      L     "MAL1S024Par".StepAct.SpeedVentilatorMaximal;
      >I    ;
      )     ; //JV160710 <=====
//BRT200310      U     "SYS_Scan0_Tick1min"
      U     "SYS_Scan0_Tick30s"; //Scan0_Tick30s
      SPBN  e614;
      L     "MAL1S024Par".Par.ParIntProcess.Value26; // Target Speed GermFan 2
      L     "MAL1S024Par".StepAct.SpeedVentilatorBasic; // linmit min
      <=I   ;
      SPB   e614;
      L     "MAL1S024Par".Par.ParIntProcess.Value26; // Target Speed GermFan 2
      L     1;
      -I    ;
      T     "MAL1S024Par".Par.ParIntProcess.Value26; // Target Speed GermFan 2
      SPA   e614;

Sum1: NOP   0;
      L     "MAL1S024Par".StepAct.SpeedVentilatorBasic;
      T     "MAL1S024Par".Par.ParIntProcess.Value26; // Target Speed GermFan 2
      U     "MAL1S024Par".Par.FlagProcess.ProcessEnd; // JV030908
      UN    "MAL1S024".PCRead.Step.StEmptying;
      UN    "MAL1S024".PCRead.Step.StEmptied;
      SPBN  e614;
      L     "MAL1S024Par".Par.ParIntProcess.Value27; // Saved Target Speed GermFan 2
      T     "MAL1S024Par".Par.ParIntProcess.Value26; // Target Speed GermFan 2
e614: NOP   0;
// store actual setpoint
      U     "MAL1S024Par".Par.FlagProcess.ProcessActive;
      U(    ;
      L     "MAL1S024Par".StepAct.SpeedVentilatorBasic;
      L     0; // setpoint recipe > 0
      >I    ;
      )     ;
      SPBN  E614;
      L     "MAL1S024Par".StepAct.SpeedVentilatorBasic;
      T     "MAL1S024Par".Par.ParIntProcess.Value27; // Saved Target Speed GermFan 2
E614: NOP   0;

NETWORK
TITLE =ASW_6050: Position waste air
//Der Betriebsart Sommerbetrieb/Winterbetrieb wird durch den Bediener per Rezept
//bestimmt.
//Wird die Kühlung im Rezept angewählt, so erfolgt die Umschaltung AUF
//Sommerbetrieb. Die Frischluftklappe wird nach dem Rezeptsollwert gestellt.
//Es erfolgt keine Regelung.
//Wird die Kühlung im Rezept abgewählt, so erfolgt die Umschaltung AUF
//Winterbetrieb. Die Frischluftklappe wird zuerst nach dem Rezeptsollwert
//gestellt. Der Rezeptsollwert ist die untere Grenze für die Regelung.
//Wird die Soll-Temperatur unter der Horde von Kühl- Heizanlage nicht eingehalten
//-Temperatur zu hoch und der Schaltpunkt überschritten, so wird die
//Frischluftklappe stufenweise geöffnet.
//Maximalwert ist 100%.
//Wird die Soll-Temperatur unter der Horde von Kühl- Heizanlage nicht eingehalten
//-Temperatur zu niedrig und der Schaltpunkt unterschritten, so wird die
//Frischluftklappe stufenweise geschlossen.
//Minimalwert ist der Rezeptsollwert.
//BRT070310 - keine AMBEV Steuerung!!!
      NOP   0;
// setpoint limit maximal position fresh air
      L     100;
      T     "MAL1S024Par".StepAct.PosFreshAirFlapMax; // limit max
      L     L#5; // 0,5°
      T     "MAL1S024Par".StepAct.DeltaTempSwitchpointAir;

// recipe setpoint
      UN(   ;
      U(    ;
      L     "MAL1S024Par".Par.ParIntMachine.ActualStep;
      L     1;
      ==I   ;
      )     ;
      UN(   ;
      L     "MAL1S024Par".Par.ProcessValue.StepTimeAct; // in ms
      L     L#1000; // in first secunde steptime
      >D    ;
      )     ;
      )     ;
// BRT17102009 - berechneter Targetwert darf nur bei StepNr.1 oder! Rezeptwert-Änderung überschrieben werden
      U(    ;
      L     "MAL1S024Par".StepAct.PosFreshAirFlapBasic;
      L     "MAL1S024Par".Par.ParIntProcess.Value24; // Rezeptwert vor Änderung
      ==D   ;
      )     ;
      SPB   Reg;
      L     "MAL1S024Par".StepAct.PosFreshAirFlapBasic;
      T     "MAL1S024Par".Par.ParIntProcess.Value24; // Rezeptwert vor Änderung

      L     "MAL1S024Par".StepAct.PosFreshAirFlapBasic;
      T     "MAL1S024Par".Par.ParIntMachine.TargetPosFreshAir;
      SPA   e605;
Reg:  NOP   0;

// Cooling or heating from cooling defive active --> no flap regulation!
//BRT030310 - Cooling angewählt in Rezept!
      U     "MAL1S024Par".Par.FlagProcess.Cooling; // request cooling
      SPB   summ;

      L     "G248M".A_2891_BTE01.OutValueUnits; //AIR TEMPERATURE BELOW FLOOR
      L     L#10; // von xx,xx°C AUF xx,x°C
      /D    ;
      L     "MAL1S024Par".StepAct.TemperaturBelowFloor;
      -D    ;
      L     "MAL1S024Par".StepAct.DeltaTempSwitchpointAir;
      >D    ;
      =     "MAL1S024Par".Par.FlagProcess1.FreshAirFlapOPEN;

      L     "G248M".A_2891_BTE01.OutValueUnits; //AIR TEMPERATURE BELOW FLOOR
      L     L#10; // von xxx,xx°C AUF xxx,x°C
      /D    ;
      L     "MAL1S024Par".StepAct.TemperaturBelowFloor;
      TAK   ;
      -D    ;
      L     "MAL1S024Par".StepAct.DeltaTempSwitchpointAir;
      >D    ;
      =     "MAL1S024Par".Par.FlagProcess1.FreshAirFlapCLOSE;

      U     "MAL1S024Par".Par.FlagProcess1.FreshAirFlapOPEN;
      U     "SYS_Scan0_Tick1min";
      SPBN  dez;
      L     "MAL1S024Par".Par.ParIntMachine.TargetPosFreshAir;
      L     "MAL1S024Par".StepAct.PosFreshAirFlapMax; // limit max
      >=I   ;
      SPB   dez;
      L     "MAL1S024Par".Par.ParIntMachine.TargetPosFreshAir;
      L     1;
      +I    ;
      T     "MAL1S024Par".Par.ParIntMachine.TargetPosFreshAir;
      SPA   e605;
dez:  NOP   0;
      U     "MAL1S024Par".Par.FlagProcess1.FreshAirFlapCLOSE;
      U     "SYS_Scan0_Tick1min";
      SPBN  e605;
      L     "MAL1S024Par".Par.ParIntMachine.TargetPosFreshAir;
      L     "MAL1S024Par".StepAct.PosFreshAirFlapBasic; // limit min
      <=I   ;
      SPB   e605;
      L     "MAL1S024Par".Par.ParIntMachine.TargetPosFreshAir;
      L     1;
      -I    ;
      T     "MAL1S024Par".Par.ParIntMachine.TargetPosFreshAir;
      SPA   e605;

summ: NOP   0;
      L     "MAL1S024Par".StepAct.PosFreshAirFlapBasic;
      T     "MAL1S024Par".Par.ParIntMachine.TargetPosFreshAir;
      SPA   e605;

e605: NOP   0;
//------------------------------------------------------------------------------------------------
//--- Position Fresh-/Recycling-Air Flap 2 ---
// recipe setpoint
      UN(   ;
      U(    ;
      L     "MAL1S024Par".Par.ParIntMachine.ActualStep;
      L     1;
      ==I   ;
      )     ;
      UN(   ;
      L     "MAL1S024Par".Par.ProcessValue.StepTimeAct; // in ms
      L     L#1000; // in first secunde steptime
      >D    ;
      )     ;
      )     ;
// BRT17102009 - berechneter Targetwert darf nur bei StepNr.1 oder! Rezeptwert-Änderung überschrieben werden
      U(    ;
      L     "MAL1S024Par".StepAct.PosFreshAirFlapBasic;
      L     "MAL1S024Par".Par.ParIntProcess.Value28; // Rezeptwert vor Änderung
      ==D   ;
      )     ;
      SPB   Reg1;
      L     "MAL1S024Par".StepAct.PosFreshAirFlapBasic;
      T     "MAL1S024Par".Par.ParIntProcess.Value28; // Rezeptwert vor Änderung

      L     "MAL1S024Par".StepAct.PosFreshAirFlapBasic;
      T     "MAL1S024Par".Par.ParIntProcess.Value29; // Target Position FreshAir 2
      SPA   e615;
Reg1: NOP   0;

// Cooling or heating from cooling defive active --> no flap regulation!
//BRT030310 - Cooling angewählt in Rezept!
      U     "MAL1S024Par".Par.FlagProcess.Cooling; // request cooling
      SPB   sum1;

      L     "G248M".A_2891_BTE03.OutValueUnits; //AIR TEMPERATURE BELOW FLOOR
      L     L#10; // von xx,xx°C AUF xx,x°C
      /D    ;
      L     "MAL1S024Par".StepAct.TemperaturBelowFloor;
      -D    ;
      L     "MAL1S024Par".StepAct.DeltaTempSwitchpointAir;
      >D    ;
      =     "MAL1S024Par".Par.FlagProcess.Inf05; // FreshAir Flap OPEN

      L     "G248M".A_2891_BTE03.OutValueUnits; //AIR TEMPERATURE BELOW FLOOR
      L     L#10; // von xxx,xx°C AUF xxx,x°C
      /D    ;
      L     "MAL1S024Par".StepAct.TemperaturBelowFloor;
      TAK   ;
      -D    ;
      L     "MAL1S024Par".StepAct.DeltaTempSwitchpointAir;
      >D    ;
      =     "MAL1S024Par".Par.FlagProcess.Inf06; // FreshAir Flap CLOSE

      U     "MAL1S024Par".Par.FlagProcess.Inf05; // FreshAir Flap OPEN
      U     "SYS_Scan0_Tick1min";
      SPBN  dez1;
      L     "MAL1S024Par".Par.ParIntProcess.Value29; // Target Position FreshAir 2
      L     "MAL1S024Par".StepAct.PosFreshAirFlapMax; // limit max
      >=I   ;
      SPB   dez1;
      L     "MAL1S024Par".Par.ParIntProcess.Value29; // Target Position FreshAir 2
      L     1;
      +I    ;
      T     "MAL1S024Par".Par.ParIntProcess.Value29; // Target Position FreshAir 2
      SPA   e615;
dez1: NOP   0;
      U     "MAL1S024Par".Par.FlagProcess.Inf06; // FreshAir Flap CLOSE
      U     "SYS_Scan0_Tick1min";
      SPBN  e615;
      L     "MAL1S024Par".Par.ParIntProcess.Value29; // Target Position FreshAir 2
      L     "MAL1S024Par".StepAct.PosFreshAirFlapBasic; // limit min
      <=I   ;
      SPB   e615;
      L     "MAL1S024Par".Par.ParIntProcess.Value29; // Target Position FreshAir 2
      L     1;
      -I    ;
      T     "MAL1S024Par".Par.ParIntProcess.Value29; // Target Position FreshAir 2
      SPA   e615;

sum1: NOP   0;
      L     "MAL1S024Par".StepAct.PosFreshAirFlapBasic;
      T     "MAL1S024Par".Par.ParIntProcess.Value29; // Target Position FreshAir 2
      SPA   e615;

e615: NOP   0;

NETWORK
TITLE =ASW_6080: Processtime Germinating
//      CALL  "SSA_MH_ProcessTime_Fct" , DB1017
//       InfDataReady :="MAL1S017".ToASW.InfDataReady
//       ProzessActive:="MAL1S017Par".Par.FlagProcess.ProcessActive
//       InStartTime  :="MAL1S017Par".Prozesstime.Starttime
//       OutStartTime :="MAL1S017Par".Prozesstime.Starttime
//       ProcessTime  :="MAL1S017Par".Prozesstime
//
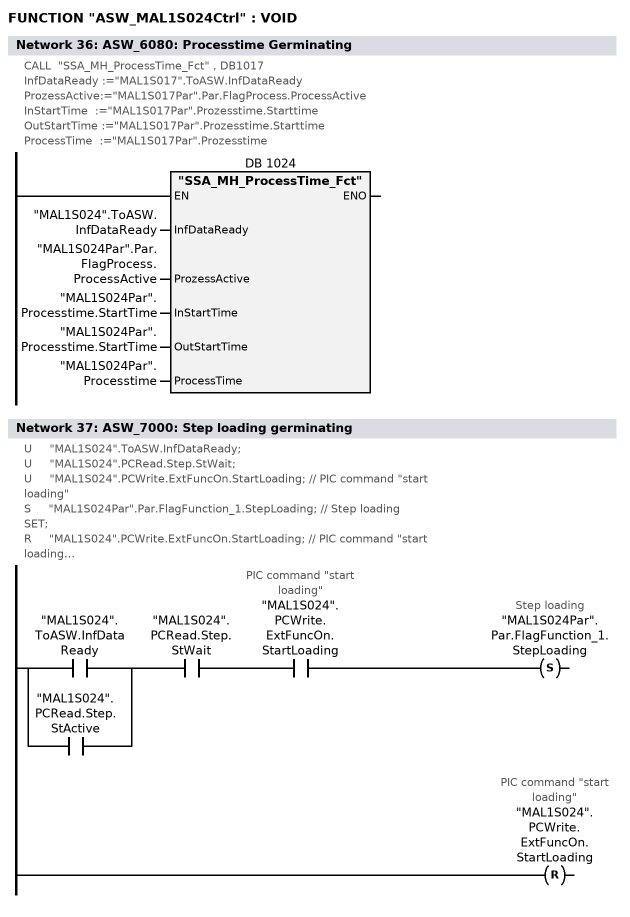

      CALL "SSA_MH_ProcessTime_Fct" , DB  1024 (
           InfDataReady             := "MAL1S024".ToASW.InfDataReady,
           ProzessActive            := "MAL1S024Par".Par.FlagProcess.ProcessActive,
           InStartTime              := "MAL1S024Par".Processtime.StartTime,
           OutStartTime             := "MAL1S024Par".Processtime.StartTime,
           ProcessTime              := "MAL1S024Par".Processtime);

NETWORK
TITLE =ASW_7000: Step loading germinating
//      U     "MAL1S024".ToASW.InfDataReady;
//      U     "MAL1S024".PCRead.Step.StWait;
//      U     "MAL1S024".PCWrite.ExtFuncOn.StartLoading; // PIC command "start
//loading"
//      S     "MAL1S024Par".Par.FlagFunction_1.StepLoading; // Step loading
//      SET;
//      R     "MAL1S024".PCWrite.ExtFuncOn.StartLoading; // PIC command "start
//loading"
////
//
//      L     WinCoS_BIW01_09PLC1BIW01_02.Ma.OutPositionAngle;
//      L     3600; // 360,0°
//      >=I   ;
//      U     "MAL1S024".ToASW.InfDataReady;
//      U     "MAL1S024".PCRead.Step.StActive;
//      U     "MAL1S024Par".Par.FlagFunction_1.StepLoading; // Step loading
//      =     "MAL1S024Par".Par.FlagFunction_1.LoadFirstPartEnd;
//
//      U     "MAL1S024".ToASW.InfDataReady;
//      U     "MAL1S024".PCRead.Step.StActive;
//      U     "MAL1S024Par".Par.FlagFunction_1.StepLoading; // Step loading
//      SPBN  E700;
//      L     "MAL1S024Par".RecipeHeader.Loading.LiftingPositionRound_1;
//      T     "MAL1S024Par".Par.ParIntProcess.NextLevelLoading; // next level
//
//      U(    ;
//      L     WinCoS_BIW01_09PLC1BIW01_02.Ma.OutPositionAngle;
//      L     "MAL1S024Par".Par.ParIntProcess.NextLevelLoading; // next level
//      >=I   ;
//      )     ;
//      O     "MAL1S024Par".Par.FlagMachine_0.Speed2ndRound;
//      SPB   Rnd2;
//      L     "MAL1S024Par".RecipeHeader.Loading.LoadingLevelRound_1;
//      T     "MAL1S024Par".Par.MachineValue.SOLLWERT_HUBZUG1_HOEHE;
//      T     "MAL1S024Par".Par.MachineValue.SOLLWERT_HUBZUG2_HOEHE;
//
//      L     "MAL1S024Par".RecipeHeader.Loading.LoadingSpeed_1;
//      T     "MAL1S024Par".Par.MachineValue.SollwertFahrantrieb;
//
//      SPA   Rnd1;
//Rnd2: NOP   0;
//      L     "MAL1S024Par".RecipeHeader.Loading.LoadingLevelRound_2;
//      T     "MAL1S024Par".Par.MachineValue.SOLLWERT_HUBZUG1_HOEHE;
//      T     "MAL1S024Par".Par.MachineValue.SOLLWERT_HUBZUG2_HOEHE;
//      L     10;
//      T     WinCoS_BIW01_09PLC1BIW01_02.Ma.Par.ParTolPosition;
//
//      L     15; // 15Hz = Wendegeschwindigkeit
//      T     "MAL1S024Par".Par.MachineValue.SollwertFahrantrieb;
//
//// Sicherheitsbit; damit bei manueller Rückwärtsfahrt über die 346°-Marke,
//nicht mit Loading Speed_0 durch den gefüllten KK gefahren wird!!
//      SET   ;
//      S     "MAL1S024Par".Par.FlagMachine_0.Speed2ndRound;
//
//Rnd1: NOP   0;
//      U  M 50.0;
//      =  M 50.0;
//      L     "MAL1S024Par".Par.ParIntMachine.TargetPosTravDriveLoad; // 450 =
//endposition loading
//      T     WinCoS_BIW01_09PLC1BIW01_02.Ma.InPositionTarget;
//E700: NOP   0;
      U     "MAL1S024".ToASW.InfDataReady;
      O     "MAL1S024".PCRead.Step.StActive;
      U     "MAL1S024".PCRead.Step.StWait;
      U     "MAL1S024".PCWrite.ExtFuncOn.StartLoading; // PIC command "start loading"
      S     "MAL1S024Par".Par.FlagFunction_1.StepLoading; // Step loading
      SET   ;
      R     "MAL1S024".PCWrite.ExtFuncOn.StartLoading; // PIC command "start loading"
//
      NOP   0;
NETWORK
TITLE =Sub 7010: Germination loading finished
//      U     "MAL1S024".ToASW.InfDataReady;
//      U     "MAL1S024".PCRead.Step.StActive;
//
//      UN    "MAL1S024".ToASW.InfSameJobPrevSec;
//      UN    "MAL1S024".PCRead.Step.StEmptying; // steep 1
//      U     "MAL1S024".PCWrite.ExtFuncOn.FinishLoading; // PIC command "finish
//loading"
//      U     "MAL1S024Par".Par.FlagFunction_1.StepLoading; // Step loading
//      S     "MAL1S024Par".Par.FlagFunction_1.FinishLoading; // loading is finish
//ed start process germinating
//      R     "MAL1S024Par".Par.FlagFunction_1.StepLoading; // Step loading
//
//      U     "MAL1S024".PCWrite.ExtFuncOn.FinishLoading; // PIC command "finish l
//oading"
//      R     "MAL1S024".PCWrite.ExtFuncOn.FinishLoading; // PIC command "finish l
//oading"
//
//      U     "MAL1S024Par".Par.FlagFunction_1.StepLoading; // Step loading
//      UN    "MAL1S024Par".Par.FlagFunction_1.FinishLoading; // loading is
//finished start process germinating
//      SPBN  save;
//      L     WinCoS_BIW01_09PLC1BIW01_02.Ma.OutPositionLeft;
//      L     WinCoS_BIW01_09PLC1BIW01_02.Ma.OutPositionRight;
//      +I    ;
//      L     2;
//      /I    ;
//      T     "MAL1S024Par".Par.ParIntMachine.LastLoadingLevel; // saved loading
//value
//save: NOP   0;
//
//      U     "MAL1S024".PCRead.Step.StReady;
//      O     "MAL1S024".PCRead.Step.StActive;
//      U     "MAL1S024Par".Par.FlagFunction_1.FinishLoading; // loading is
//finished start process germinating
//      UN     "MAL1S024Par".Par.FlagFunction_1.StepLoading; // Step loading
//      R     "MAL1S024Par".Par.FlagMachine_0.Speed2ndRound;
//fin:  NOP   0;
//E701: NOP   0;
// Previous Section always the Sec.801
///
      L     "MAL1S024".ToSSW.InPrevSecDB;
      L     0;
      <>I   ;
      SPB   prev;
      L     801;
      T     "MAL1S024".ToSSW.InPrevSecDB;
prev: NOP   0;

      U     "MAL1S024".ToASW.InfDataReady;
      U     "MAL1S024".PCRead.Step.StActive;
      UN    "MAL1S024".PCRead.Step.StEmptying; //
      U     "MAL1S024".PCWrite.ExtFuncOn.FinishLoading; // PIC command "finish loading"
      U     "MAL1S024Par".Par.FlagFunction_1.StepLoading; // Step loading
      O(    ;
      UN    "MAL1S024".SecNom.Par1On.Cmd01; // With Loading
      UN    "MAL1S024".ToASW.InfSameBatchPrevSec;
      U     "MAL1S024".ToASW.InfDataReady;
      U     "MAL1S024".PCRead.Step.StActive;
      )     ;
      S     "MAL1S024Par".Par.FlagFunction_1.FinishLoading; // loading is finished start process germinating
      R     "MAL1S024Par".Par.FlagFunction_1.StepLoading; // Step loading

      U     "MAL1S024".PCWrite.ExtFuncOn.FinishLoading; // PIC command "finish loading"
      R     "MAL1S024".PCWrite.ExtFuncOn.FinishLoading; // PIC command "finish loading"


      U     "MAL1S024".PCRead.Step.StReady;
      O     "MAL1S024".PCRead.Step.StActive;
      U     "MAL1S024Par".Par.FlagFunction_1.FinishLoading; // loading is finished start process germinating
      UN    "MAL1S024Par".Par.FlagFunction_1.StepLoading; // Step loading
      R     "MAL1S024Par".Par.FlagMachine_0.Speed2ndRound;
      NOP   0;
      NOP   0;
NETWORK
TITLE =ASW_8000:  Step unloading germination
//      U     "MAL1S024".ToASW.InfDataReady
//      U     "MAL1S024".PCRead.Step.StEmptying
//      U     "MAL1S024".ToASW.InfSameJobNextSec
//      UN    "MAL1S024Par".Par.FlagFunction_1.StepUnloading    // Step unloading
//      UN    "MAL1S024Par".Par.FlagFunction_1.FinishUnloading
//      U     "MAL1S024Par".Par.FlagMachine_0.CouplingDischargFinished
//      U     "MAL1S024Par".Par.FlagMachine_0.WallUnCoupled
//      S     "MAL1S024Par".Par.FlagFunction_1.StepUnloading    // Step unloading
//
//      U     "MAL1S024Par".Par.FlagFunction_1.StepUnloading    // Step unloading
//      U     "MAL1S024Par".Par.FlagFunction_1.UnloadingStarted
//      U     "MAL1S024".ToASW.spare34    // infNextSectionFeeding
//      =     "MAL1S024Par".Par.FlagFunction_0.InfReleaseUnloading    // from
//kiln
//
//      U     "MAL1S024Par".Par.FlagFunction_1.StepUnloading    // Step unloading
//      UN    "MAL1S024Par".Par.FlagFunction_1.UnloadingStarted
//      U     "G242M".A_2815_BZS22.StFalse    // backwall is not in down pos
//      U     "G242M".A_2815_BZS23.StTrue // backwall is in up pos  // JV030908
//      U     "G247M".A_2811_KCL01I5.StTrue    // pushbutton drive fast fwd
//      S     "MAL1S024Par".Par.FlagFunction_1.UnloadingStarted
//      FP    "MAL1S024Par".Par.FlagFunction_0.FlagUnloadingStartedFP    //
//JV030908
//      =     "MAL1S024Par".Par.FlagFunction_0.ImpulseUnloadingStarted    //
//JV030908
//
//      UN    "MAL1S024Par".Par.FlagFunction_1.UnloadingStarted
//      O     "MAL1S024Par".Par.FlagFunction_1.StepCleaning    // Step cleaning
//      O     "MAL1S024Par".Par.FlagFunction_1.FinishCleaning
//      SPB   EN38
//      L     3600
//      T     "G245M".A_2811_MXZ41MA.Ma.InPositionTarget    // target position
//unloading
//      L     "MAL1S024Par".RecipeHeader.Unloading.UnLoadingSpeed_2    // JV
//290808
//      T     "MAL1S024Par".Par.ParIntProcess.CopyLoadindSpeed2    // JV 290808
//EN38: NOP   0
//
      U     "MAL1S024".ToASW.InfDataReady;
      U     "MAL1S024".PCRead.Step.StEmptying;
//====>BRT070310
      U(    ;
      O     "MAL1S024".ToASW.InfSameJobNextSec;
      O(    ;
      L     831; // Next Section: MAL1S031
      L     "MAL1S024".SecNom.HEADER.Kilning_vessel_1; // Target in recipe
      ==I   ;
      )     ;
      )     ;
//<====BRT070310
      UN    "MAL1S024Par".Par.FlagFunction_1.StepUnloading; // Step unloading
      UN    "MAL1S024Par".Par.FlagFunction_1.FinishUnloading;
      U     "MAL1S024Par".Par.FlagMachine_0.CouplingDischargFinished;
      U     "MAL1S024Par".Par.FlagMachine_0.WallUnCoupled;
//BRT070310 - Start Unloading Button vergessen
      U     "MAL1S024".PCWrite.ExtFuncOn.StartUnLoading; // PIC command "Start Unloading"
      S     "MAL1S024Par".Par.FlagFunction_1.StepUnloading; // Step unloading

//BRT070310 - Start Unloading Button vergessen
      U     "MAL1S024".PCWrite.ExtFuncOn.StartUnLoading; // PIC command "Start Unloading"
      R     "MAL1S024".PCWrite.ExtFuncOn.StartUnLoading; // PIC command "Start Unloading"

      U     "MAL1S024Par".Par.FlagFunction_1.StepUnloading; // Step unloading
      U     "MAL1S024Par".Par.FlagFunction_1.UnloadingStarted;
//====>BRT070310
      U(    ;
      O     "MAL1S024".ToASW.spare34; // infNextSectionFeeding
      O(    ;
      L     831; // Next Section: MAL1S031
      L     "MAL1S024".SecNom.HEADER.Kilning_vessel_1; // Target in recipe
      ==I   ;
      )     ;
      )     ;
//<====BRT070310
      =     "MAL1S024Par".Par.FlagFunction_0.InfReleaseUnloading; // from kiln

      U     "MAL1S024Par".Par.FlagFunction_1.StepUnloading; // Step unloading
      UN    "MAL1S024Par".Par.FlagFunction_1.UnloadingStarted;
      U     "G242M".A_2815_BZS22.StFalse; // backwall is not in down pos
      U     "G242M".A_2815_BZS23.StTrue; // backwall is in up pos  // JV030908
      U     "G247M".A_2811_KCL01I5.StTrue; // pushbutton drive fast fwd
      S     "MAL1S024Par".Par.FlagFunction_1.UnloadingStarted;
      FP    "MAL1S024Par".Par.FlagFunction_0.FlagUnloadingStartedFP; // JV030908
      =     "MAL1S024Par".Par.FlagFunction_0.ImpulseUnloadingStarted; // JV030908

      UN    "MAL1S024Par".Par.FlagFunction_1.UnloadingStarted;
      O     "MAL1S024Par".Par.FlagFunction_1.StepCleaning; // Step cleaning
      O     "MAL1S024Par".Par.FlagFunction_1.FinishCleaning;
      SPB   EN38;
//BRT250310      L     3600
      L     4000; //BRT250310 -> +2° Overlapping damit die Maschine sicher auf den Endschalter fährt!
      T     "G245M".A_2811_MXZ41MA.Ma.InPositionTarget; // target position unloading
      L     "MAL1S024Par".RecipeHeader.Unloading.UnLoadingSpeed_2; // JV 290808
      T     "MAL1S024Par".Par.ParIntProcess.CopyLoadindSpeed2; // JV 290808
EN38: NOP   0;

NETWORK
TITLE =ASW_8010:  Step unloading finished
//// Verweilzeit auf dem Endschalter  =A_2111_BZS44.StTrue --> stop discharge side
//      L     S5T#10M                     // Verweilzeit auf dem Endschalter
//      U     "G245M".A_2811_BZS44.StTrue // stop discharge side
//      U     "G244M".A_2815_BZS42.StTrue
//      SE    T    123
////******************************************************************************
//******************
//
//      U     "MAL1S024".ToASW.InfDataReady
//      U     "MAL1S024".PCRead.Step.StEmptying
//      U     "MAL1S024".ToASW.InfSameJobNextSec
//      U     "MAL1S024Par".Par.FlagFunction_1.StepUnloading    // Step unloading
//      UN    "MAL1S024Par".Par.FlagFunction_1.FinishUnloading
//      U     "MAL1S024Par".Par.FlagFunction_1.StepUnloading    // Step unloading
//      U     "MAL1S024Par".Par.FlagFunction_1.UnloadingStarted
//      U     T    123                    // Verweilzeit auf dem Endschalter ist
//abgelaufen
////------------ Confirmation is necessary to finish unloading
//**********************
//      U(
//      L     "G245M".A_2811_MXZ41MA.Ma.OutPositionRel
//      L     950                         //95%
//      >I
//      )
////      U     "MAL1S024".PCWrite.ExtFuncOn.FinishCleanSurface    // PIC command
//"Finish Unloading"
////******************************************************************************
//******************
//      R     "MAL1S024Par".Par.FlagFunction_1.StepUnloading    // Step unloading
//      S     "MAL1S024Par".Par.FlagFunction_1.FinishUnloading
//      S     "MAL1S024Par".Par.FlagMachine_0.CmdTurnRevAfterUnloading
//      UN    "MAL1S024Par".Par.FlagMachine_0.CmdTurnRevAfterUnloading
//      SPB   EN39
//      L     3399
//      T     "G245M".A_2811_MXZ41MA.Ma.InPositionTarget    // target position
//EN39: NOP   0
//
//      SET
//      R     "MAL1S024".PCWrite.ExtFuncOn.FinishCleanSurface    // PIC command
//"Finish Unloading"
//
// Verweilzeit auf dem Endschalter  =A_2811_BZS44.StTrue --> stop discharge side
//      L     S5T#5M                      // Verweilzeit auf dem Endschalter
//BRT070310      U     "G245M".A_2811_BZS44.StTrue // stop discharge side
      U     "G245M".A_2811_BZS46.StTrue; // stop endposition unloading
//BRT070310      U     "G244M".A_2815_BZS42.StTrue
      U     "G246M".A_2815_MXZ11MA.Ma.StStartedFwd;
//      SE    T    124
//====>BRT070410 - ohne Timer, um Restart der Wartezeit bei Unterbruch Transport zu verhindern!
      UN    "MAL1S024Par".Par.FlagFunction_0.Inf29; //Wartezeit 300s abgelaufen = 1
      U     "SYS_Scan0_Tick1s";
      SPBN  wait;
      L     "MAL1S024Par".Par.ParIntMachine.Value33; //aktuelle Wartezeit Maschine bei 100% Unloading-Position
      L     1;
      +I    ;
      T     "MAL1S024Par".Par.ParIntMachine.Value33; //aktuelle Wartezeit Maschine bei 100% Unloading-Position
wait: NOP   0;
      L     "MAL1S024Par".Par.ParIntMachine.Value33; //aktuelle Wartezeit Maschine bei 100% Unloading-Position
      L     300; // 300s
      >=I   ;
      =     "MAL1S024Par".Par.FlagFunction_0.Inf29; //Wartezeit 300s abgelaufen = 1
//<====BRT070410
//************************************************************************************************

      U     "MAL1S024".ToASW.InfDataReady;
      U     "MAL1S024".PCRead.Step.StEmptying;
//====>BRT070310
      U(    ;
      O     "MAL1S024".ToASW.InfSameJobNextSec;
      O(    ;
      L     831; // Next Section: MAL1S031
      L     "MAL1S024".SecNom.HEADER.Kilning_vessel_1; // Target in recipe
      ==I   ;
      )     ;
      )     ;
//<====BRT070310
      U     "MAL1S024Par".Par.FlagFunction_1.StepUnloading; // Step unloading
      UN    "MAL1S024Par".Par.FlagFunction_1.FinishUnloading;
      U     "MAL1S024Par".Par.FlagFunction_1.StepUnloading; // Step unloading
      U     "MAL1S024Par".Par.FlagFunction_1.UnloadingStarted;
//      U     T    124                    // Verweilzeit auf dem Endschalter ist abgelaufen
      U(    ;
      U     "MAL1S024Par".Par.FlagFunction_0.Inf29; //Wartezeit 300s abgelaufen = 1
      O     "MAL1S024".PCWrite.ExtFuncOn.FinishCleanSurface; // PIC command "Finish Unloading"
      )     ;
//------------ Confirmation is necessary to finish unloading **********************
      U(    ;
      L     "G245M".A_2811_MXZ41MA.Ma.OutPositionRel;
      L     950; //95%
      >I    ;
      )     ;
//      U     "MAL1S024".PCWrite.ExtFuncOn.FinishCleanSurface    // PIC command "Finish Unloading"
//************************************************************************************************
      R     "MAL1S024Par".Par.FlagFunction_1.StepUnloading; // Step unloading
      S     "MAL1S024Par".Par.FlagFunction_1.FinishUnloading;
      S     "MAL1S024Par".Par.FlagMachine_0.CmdTurnRevAfterUnloading;
      S     "MAL1S024Par".Par.FlagGen.Flag0024; // finished first unloading
      UN    "MAL1S024Par".Par.FlagMachine_0.CmdTurnRevAfterUnloading;
      SPB   EN39;
      L     3399;
      T     "G245M".A_2811_MXZ41MA.Ma.InPositionTarget; // target position
EN39: NOP   0;

NETWORK
TITLE =ASW_9000: Step cleaning germination box
//
      U     "MAL1S024".ToASW.InfDataReady;
      U(    ;
      U     "MAL1S024".PCRead.Step.StEmptied;
      O     "MAL1S024".PCRead.Step.StEmptying;
      )     ;
      U     "MAL1S024Par".Par.FlagFunction_1.FinishUnloading;
      U     "MAL1S024Par".Par.FlagMachine_0.CmdTurnRevAfterUnloading;
      UN    "MAL1S024Par".Par.FlagMachine_0.CleaningAfterUnloading;
      U(    ;
      L     "G245M".A_2811_MXZ41MA.Ma.OutPositionRel;
      L     956;
      <=I   ; // cleaning pos
      )     ;
      U     "G245M".A_2811_BZS46.StFalse; // stop endposition unloading //JV040310
      U     "MAL1S024Par".Par.FlagGen.Flag0024; // finished first unloading
      UN    "MAL1S024Par".Par.FlagGen.Flag0025; // wait pos. to unloading leftover
      UN    "MAL1S024Par".Par.FlagGen.Flag0026; // unloading leftover
      UN    "MAL1S024Par".Par.FlagGen.Flag0027; // finished unloading leftover
      O     "MAL1S024".PCWrite.ExtFuncOn.FinishCleanSurface; // PIC command "Finish Unloading"
      R     "MAL1S024Par".Par.FlagMachine_0.CmdTurnRevAfterUnloading;
      R     "MAL1S024Par".Par.FlagGen.Flag0024; // finished first unloading
      S     "MAL1S024Par".Par.FlagGen.Flag0025; // wait pos. to unloading leftover

//--- Zwischenschritt für Starten einer Restentladung ---
      U     "G247M".A_2811_KCL01I5.StTrue; // pushbutton drive fast fwd
      UN    "MAL1S024Par".Par.FlagGen.Flag0024; // finished first unloading
      U     "MAL1S024Par".Par.FlagGen.Flag0025; // wait pos. to unloading leftover
      UN    "MAL1S024Par".Par.FlagGen.Flag0026; // unloading leftover
      U(    ;
      U     "MAL1S024".PCRead.Step.StEmptied;
      O     "MAL1S024".PCRead.Step.StEmptying;
      )     ;
      U     "MAL1S024Par".Par.FlagFunction_1.FinishUnloading;
      UN    "MAL1S024Par".Par.FlagMachine_0.CmdTurnRevAfterUnloading;
      UN    "MAL1S024Par".Par.FlagMachine_0.CleaningAfterUnloading;
      U(    ;
      L     "G245M".A_2811_MXZ41MA.Ma.OutPositionRel;
      L     956;
      <=I   ; // cleaning pos
      )     ;
      U     "G245M".A_2811_BZS46.StFalse; // stop endposition unloading
      O     "MAL1S024".PCWrite.ExtFuncOn.FinishCleanSurface; // PIC command "Finish Unloading"
      R     "MAL1S024Par".Par.FlagMachine_0.CmdTurnRevAfterUnloading;
      R     "MAL1S024Par".Par.FlagGen.Flag0025; // wait pos. to unloading leftover
      S     "MAL1S024Par".Par.FlagGen.Flag0026; // unloading leftover

      UN    "MAL1S024Par".Par.FlagGen.Flag0026; // unloading leftover
      SPB   EN40;
      L     4000;
      T     "G245M".A_2811_MXZ41MA.Ma.InPositionTarget; // target position
EN40: NOP   0;

//--- Erreichen der Endposition nach Restentladung ---
      U     "G245M".A_2811_BZS46.StTrue; // stop endposition unloading
      U     "MAL1S024Par".Par.FlagFunction_1.FinishUnloading;
      U     "MAL1S024Par".Par.FlagGen.Flag0026; // unloading leftover
      U(    ;
      L     "G245M".A_2811_MXZ41MA.Ma.OutPositionRel;
      L     950; //95%
      >I    ;
      )     ;
      O     "MAL1S024".PCWrite.ExtFuncOn.FinishCleanSurface; // PIC command "Finish Unloading"
      R     "MAL1S024Par".Par.FlagGen.Flag0026; // unloading leftover
      S     "MAL1S024Par".Par.FlagGen.Flag0027; // finished unloading leftover
      S     "MAL1S024Par".Par.FlagMachine_0.CmdTurnRevAfterUnloading;

//********************************************************************************************

      U     "MAL1S024".ToASW.InfDataReady;
//====>BRT040310
      U(    ;
      U     "MAL1S024".PCRead.Step.StEmptied;
      O     "MAL1S024".PCRead.Step.StEmptying;
      )     ;
//<====BRT040310
      U     "MAL1S024Par".Par.FlagFunction_1.FinishUnloading;
      U     "MAL1S024Par".Par.FlagMachine_0.CmdTurnRevAfterUnloading;
      UN    "MAL1S024Par".Par.FlagMachine_0.CleaningAfterUnloading;
      U(    ;
      L     "G245M".A_2811_MXZ41MA.Ma.OutPositionRel;
      L     956;
      <=I   ; // cleaning pos
      )     ;
      U     "G245M".A_2811_BZS46.StFalse; // stop endposition unloading //JV040310
//====>BRT120510
      UN    "MAL1S024Par".Par.FlagGen.Flag0024; // finished first unloading
      UN    "MAL1S024Par".Par.FlagGen.Flag0025; // wait pos. to unloading leftover
      UN    "MAL1S024Par".Par.FlagGen.Flag0026; // unloading leftover
      U     "MAL1S024Par".Par.FlagGen.Flag0027; // finished unloading leftover
      O     "MAL1S024".PCWrite.ExtFuncOn.FinishCleanSurface; // PIC command "Finish Unloading"
      R     "MAL1S024Par".Par.FlagGen.Flag0027; // finished unloading leftover
//<====BRT120510
      R     "MAL1S024Par".Par.FlagMachine_0.CmdTurnRevAfterUnloading;
      R     "MAL1S024Par".Par.FlagFunction_1.FinishUnloading;
      S     "MAL1S024Par".Par.FlagMachine_0.CleaningAfterUnloading;
      S     "MAL1S024Par".Par.FlagFunction_1.StepCleaning; // Step cleaning

      SET   ;
      R     "MAL1S024".PCWrite.ExtFuncOn.FinishCleanSurface; // PIC command "Finish Unloading"

NETWORK
TITLE =ASW_9010: Cleaning Germination box finished
//
      U     "MAL1S024".ToASW.InfDataReady;
//====>BRT070310
      U(    ;
      U     "MAL1S024".PCRead.Step.StEmptied;
      O     "MAL1S024".PCRead.Step.StEmptying;
      )     ;
//<====BRT070310
      U     "MAL1S024Par".Par.FlagFunction_1.StepCleaning; // Step cleaning
      U     "G245M".A_2811_BZS44.StFalse; // stop discharge side
      U(    ;
      O     "MAL1S024".PCWrite.ExtFuncOn.FinishCleaning; // PIC command "cleaning finished"
// BRT110310      O     "G247M".A_2811_KCL01I4.InpTrue    // pushbutton "drive rev"
      O     "G247M".A_2811_KCL01I6.InpTrue; // pushbutton "drive rev fast"
      )     ;
      R     "MAL1S024Par".Par.FlagMachine_0.CleaningAfterUnloading;
      R     "MAL1S024Par".Par.FlagFunction_1.StepCleaning; // Step cleaning
      S     "MAL1S024Par".Par.FlagFunction_1.FinishCleaning;

      SET   ;
      R     "MAL1S024".PCWrite.ExtFuncOn.FinishCleaning; // PIC command "cleaning finished"

      U     "MAL1S024".PCRead.Step.StIdling;
//BRT070310      U     "G245M".A_2811_BZS46.StTrue // stop fan side (home pos)
      U     "G245M".A_2811_BZS44.StTrue; // stop zeroposition (home pos)
      U(    ; //dyk 081031 50 pulses
      L     "G245M".A_2811_MXZ41MA.IncCounter.InpActCount;
      L     50;
      <I    ;
      )     ;
      R     "MAL1S024Par".Par.FlagFunction_1.FinishCleaning;

      UN    "MAL1S024Par".Par.FlagFunction_1.FinishCleaning;
      SPB   EN41;
      L     0;
      T     "G245M".A_2811_MXZ41MA.Ma.InPositionTarget; // target position
//MW 2008.10.24
      L     "MAL1S024Par".RecipeHeader.Unloading.UnLoadingSpeed_2;
      T     "MAL1S024Par".Par.ParIntProcess.CopyLoadindSpeed2;
EN41: NOP   0;

NETWORK
TITLE =ASW_9080: Send section date to PIC after germination

      AUF   "MAL1S024";
      U     "MAL1S024".PCRead.Step.StEmptying;
      FP    "MAL1S024Par".Par.FlagProcess.FP_SendResultToPIC;
      SPBN  E908;
//

E908: NOP   0;
NETWORK
TITLE =ASW_10000: ILO functions

      U     "MAL1S024".SecAc.Sta1On.Inf08;
      =     "MAL1S024".Gr.All.Spare04;

// reset ILO with start unloading   JV080908    special on SALADIN BOXES
      U     "MAL1S024Par".Par.FlagFunction_0.ImpulseUnloadingStarted; // JV030908
      R     "MAL1S024".SecAc.Sta1On.Inf08;

//- Little help for PIC-People
      U     "MAL1S024".SecAc.Sta1On.Inf08;
      SPB   RSM;
      L     0;
      T     "MAL1S024Par".Ilo.Code_ILO_Funktion0; // FCM 24 LINE 1 SEC 24  GERM 8
RSM:  NOP   0;
//- Combination OLD and NEW ---
      U     "MAL1S024".SecAc.Sta1On.Inf08;
      SPBN  IFM;
      L     "MAL1S024Par".Ilo.ILOMode;
      L     100;
      *I    ;
      T     "MAL1S024Par".Ilo.Code_ILO_Funktion0;
IFM:  NOP   0;

//  no ILO-mode >> cmd manual off to all used groups and reset all flags
      U     "MAL1S024".SecAc.Sta1On.Inf08;
      FN    "MAL1S024Par".Ilo.Flag.EdgeILOModeOn; //BRT070310
//BRT070310      FN    DB910.DBX 3692.0
//      S     DB909.DBX 3006.0            // (ManOff)
//      R     DB909.DBX 3014.0
//      R     DB909.DBX 3018.1
//  Gr-cmd manual OFF
      S     "G014G".Gr.CmdManualOff; // GENERAL ELEMENTS GERM 8
      S     "G242M".Gr.CmdManualOff; // LIFTING DEVICE  GERM 8
      S     "G243M".Gr.CmdManualOff; // COUPLING DEVICE TURNER  GERM 8
      S     "G244M".Gr.CmdManualOff; // COUPLING DEVICE WALL  GERM 8
      S     "G245M".Gr.CmdManualOff; // TRAVELLING DRIVE  GERM 8
      S     "G246M".Gr.CmdManualOff; // HORIZONTAL AND LIFTING SCREW  GERM 8
      S     "G249M".Gr.CmdManualOff; // TURNING SCREWS  GERM 8
      S     "G250M".Gr.CmdManualOff; // FAN AND VALVE SRAY AIR  GERM 8
      S     "G251M".Gr.CmdManualOff; // FRESH AIR LOUVER  GERM 8
      S     "G252M".Gr.CmdManualOff; // EXHAUST AIR LOUVER  GERM 8
      S     "G257M".Gr.CmdManualOff; // COOLING / HEATING  GERM 8
//  RESET ADDITIONAL CMD`S
      R     "G242M".USW14; // ILO-cmd
      R     "G242M".USW15; // ILO-cmd
      R     "G243M".USW14; // ILO-cmd
      R     "G243M".USW15; // ILO-cmd
      R     "G244M".USW14; // ILO-cmd
      R     "G244M".USW15; // ILaO-cmd
      R     "G245M".USW14; // ILO-cmd
      R     "G245M".USW15; // ILO-cmd
      R     "G246M".USW14; // ILO-cmd
      R     "G246M".USW15; // ILO-cmd
      R     "G249M".USW14; // ILO-cmd
      R     "G249M".USW15; // ILO-cmd
      R     "G250M".USW14; // ILO-cmd
      R     "G250M".USW15; // ILO-cmd
      R     "G251M".USW14; // ILO-cmd
      R     "G251M".USW15; // ILO-cmd
      R     "G252M".USW14; // ILO-cmd
      R     "G252M".USW15; // ILO-cmd
      R     "G257M".USW14; // ILO-cmd
      R     "G257M".USW15; // ILO-cmd

      U     "MAL1S024".SecAc.Sta1On.Inf08;
      SPB   RSM2;
      L     0;
      T     #tmpInt;
      CALL "SIEMENS_FILL" (
           BVAL                     := #tmpInt,
           RET_VAL                  := #tmpRET,
           BLK                      := "MAL1S024Par".Ilo);
RSM2: NOP   0;

      NOP   0;
// --- FCM 04 - Fans ---
      L     "MAL1S024Par".Ilo.ILOMode;
      L     4;
      <>I   ;
      SPB   IO4;
// man on
      U     "MAL1S024Par".Ilo.GrCMDManOn[1];
      S     "G250M".Gr.InManual; // FAN AND VALVE SRAY AIR  GERM 8
      S     "G251M".Gr.InManual; // FRESH AIR LOUVER  GERM 8
      S     "G252M".Gr.InManual; // EXHAUST AIR LOUVER  GERM 8
      R     "MAL1S024Par".Ilo.GrCMDManOn[1];
// man off
      U     "MAL1S024Par".Ilo.GrCMDManOff[1];
      S     "G250M".Gr.CmdManualOff; // FAN AND VALVE SRAY AIR  GERM 8
      R     "G250M".Gr.InManual; // FAN AND VALVE SRAY AIR  GERM 8
      R     "G250M".USW14; // ILO-cmd
      R     "G250M".USW15; // ILO-cmd
      S     "G251M".Gr.CmdManualOff; // FRESH AIR LOUVER  GERM 8
      R     "G251M".Gr.InManual; // FRESH AIR LOUVER  GERM 8
      R     "G251M".USW14; // ILO-cmd
      R     "G251M".USW15; // ILO-cmd
      S     "G252M".Gr.CmdManualOff; // EXHAUST AIR LOUVER  GERM 8
      R     "G252M".Gr.InManual; // EXHAUST AIR LOUVER  GERM 8
      R     "G252M".USW14; // ILO-cmd
      R     "G252M".USW15; // ILO-cmd
      R     "MAL1S024Par".Ilo.GrCMDManOff[1];
      R     "MAL1S024Par".Ilo.GrCMDManAdditional.Cmd1[1];
      R     "MAL1S024Par".Ilo.GrCMDManAdditional.Cmd2[1];
// man start
      U     "MAL1S024Par".Ilo.GrCMDManStart[1];
      S     "G250M".Gr.CmdOn; // FAN AND VALVE SRAY AIR  GERM 8
      S     "G250M".Gr.CmdContinue; // FAN AND VALVE SRAY AIR  GERM 8
      S     "G251M".Gr.CmdOn; // FRESH AIR LOUVER  GERM 8
      S     "G251M".Gr.CmdContinue; // FRESH AIR LOUVER  GERM 8
      S     "G252M".Gr.CmdOn; // EXHAUST AIR LOUVER  GERM 8
      S     "G252M".Gr.CmdContinue; // EXHAUST AIR LOUVER  GERM 8
      R     "MAL1S024Par".Ilo.GrCMDManStart[1];
      U     "MAL1S024Par".Ilo.GrCMDManStart[2];
      R     "MAL1S024Par".Ilo.GrCMDManStart[2];
// man stop
      U     "MAL1S024Par".Ilo.GrCMDManStop[1];
      S     "G250M".Gr.CmdOff; // FAN AND VALVE SRAY AIR  GERM 8
//BRT070310      S     "G250M".Gr.CmdOff           // FRESH AIR LOUVER  GERM 8
//BRT070310      S     "G250M".Gr.CmdOff           // EXHAUST AIR LOUVER  GERM 8
      R     "MAL1S024Par".Ilo.GrCMDManStop[1];
// man fault reset
//BRT070310      U     "MAL1S024Par".Ilo.GrCMDManOn[17]
      U     "MAL1S024Par".Ilo.GrCMDManFaultReset[1]; //BRT070310
      S     "G250M".Gr.CmdFaultReset; // FAN AND VALVE SRAY AIR  GERM 8
      S     "G251M".Gr.CmdFaultReset; // FRESH AIR LOUVER  GERM 8
      S     "G252M".Gr.CmdFaultReset; // EXHAUST AIR LOUVER  GERM 8
      R     "MAL1S024Par".Ilo.GrCMDManFaultReset[1]; //BRT070310
// target position
      UN    "G250M".Gr.InManual; // FAN AND VALVE SRAY AIR  GERM 8
      O(    ;
      L     "MAL1S024Par".Ilo.Code_ILO_Funktion0;
      L     400;
      <>I   ;
      )     ;
      SPB   F04a;
      L     "MAL1S024Par".Ilo.SetpointInt01[1];
      T     "MAL1S024Par".Par.ParIntProcess.Speed_ILO_Fan;
F04a: NOP   0;
//BRT070310 - Sollwert Frischluftklappen!
      UN    "G251M".Gr.InManual; // FRESH AIR LOUVER GERM 8
      O(    ;
      L     "MAL1S024Par".Ilo.Code_ILO_Funktion0;
      L     400;
      <>I   ;
      )     ;
      SPB   F04b;
      L     "MAL1S024Par".Ilo.SetpointInt02[1];
      T     "MAL1S024Par".Par.ParIntProcess.TarPos_ILO_FreshAir;
F04b: NOP   0;

IO4:  NOP   0;
      NOP   0;
// --- FCM 05 - Fans with target air temperature ---
      L     "MAL1S024Par".Ilo.ILOMode;
      L     5;
      <>I   ;
      SPB   IO5;
// man on
      U     "MAL1S024Par".Ilo.GrCMDManOn[1];
      S     "G250M".Gr.InManual; // FAN AND VALVE SRAY AIR  GERM 8
      S     "G251M".Gr.InManual; // FRESH AIR LOUVER  GERM 8
      S     "G257M".Gr.InManual; // COOLING / HEATING  GERM 8
      S     "G252M".Gr.InManual; // EXHAUST AIR LOUVER GERM 8  //BRT070310
      R     "MAL1S024Par".Ilo.GrCMDManOn[1];
// man off
      U     "MAL1S024Par".Ilo.GrCMDManOff[1];
      S     "G250M".Gr.CmdManualOff; // FAN AND VALVE SRAY AIR  GERM 8
      R     "G250M".Gr.InManual; // FAN AND VALVE SRAY AIR  GERM 8
      R     "G250M".USW14; // ILO-cmd
      R     "G250M".USW15; // ILO-cmd
      S     "G251M".Gr.CmdManualOff; // FRESH AIR LOUVER  GERM 8
      R     "G251M".Gr.InManual; // FRESH AIR LOUVER  GERM 8
      R     "G251M".USW14; // ILO-cmd
      R     "G251M".USW15; // ILO-cmd
      S     "G257M".Gr.CmdManualOff; // COOLING / HEATING  GERM 8
      R     "G257M".Gr.InManual; // COOLING / HEATING  GERM 8
      R     "G257M".USW14; // ILO-cmd
      R     "G257M".USW15; // ILO-cmd
      S     "G252M".Gr.CmdManualOff; // EXHAUST AIR LOUVER GERM 8  //BRT070310
      R     "G252M".Gr.InManual; // EXHAUST AIR LOUVER GERM 8  //BRT070310
      R     "G252M".USW14; // ILO-cmd                    //BRT070310
      R     "G252M".USW15; // ILO-cmd                    //BRT070310
      R     "MAL1S024Par".Ilo.GrCMDManOff[1];
      R     "MAL1S024Par".Ilo.GrCMDManAdditional.Cmd1[1];
      R     "MAL1S024Par".Ilo.GrCMDManAdditional.Cmd2[1];
// man start
      U     "MAL1S024Par".Ilo.GrCMDManStart[1];
      S     "G250M".Gr.CmdOn; // FAN AND VALVE SRAY AIR  GERM 8
      S     "G250M".Gr.CmdContinue; // FAN AND VALVE SRAY AIR  GERM 8
      S     "G251M".Gr.CmdOn; // FRESH AIR LOUVER  GERM 8
      S     "G251M".Gr.CmdContinue; // FRESH AIR LOUVER  GERM 8
      S     "G257M".Gr.CmdOn; // COOLING / HEATING  GERM 8
      S     "G257M".Gr.CmdContinue; // COOLING / HEATING  GERM 8
      S     "G252M".Gr.CmdOn; // EXHAUST AIR LOUVER GERM 8   //BRT070310
      S     "G252M".Gr.CmdContinue; // EXHAUST AIR LOUVER GERM 8   //BRT070310
      R     "MAL1S024Par".Ilo.GrCMDManStart[1];
      U     "MAL1S024Par".Ilo.GrCMDManStart[2];
      R     "MAL1S024Par".Ilo.GrCMDManStart[2];
// man stop
      U     "MAL1S024Par".Ilo.GrCMDManStop[1];
      S     "G250M".Gr.CmdOff; // FAN AND VALVE SRAY AIR  GERM 8
//BRT070310      S     "G251M".Gr.CmdOff           // FRESH AIR LOUVER GERM 8
//BRT070310      S     "G252M".Gr.CmdOff           // EXHAUST AIR LOUVER GERM 8
      S     "G257M".Gr.CmdOff; // COOLING / HEATING  GERM 8
      R     "MAL1S024Par".Ilo.GrCMDManStop[1];
// man fault reset
      U     "MAL1S024Par".Ilo.GrCMDManFaultReset[1];
      S     "G250M".Gr.CmdFaultReset; // FAN AND VALVE SRAY AIR  GERM 8
      S     "G251M".Gr.CmdFaultReset; // FRESH AIR LOUVER  GERM 8
      S     "G257M".Gr.CmdFaultReset; // COOLING / HEATING  GERM 8
      S     "G252M".Gr.CmdFaultReset; // EXHAUST AIR LOUVER GERM 8   //BRT070310
      R     "MAL1S024Par".Ilo.GrCMDManFaultReset[1];
// target position
      UN    "G257M".Gr.InManual; // COOLING / HEATING  GERM 8
      SPB   F05a;
      L     "MAL1S024Par".Ilo.SetpointInt02[1];
      T     "MAL1S024Par".Par.ParIntProcess.TargetTemperature_ILO;
F05a: NOP   0;
      UN    "G250M".Gr.InManual; // FAN AND VALVE SRAY AIR  GERM 8
      O(    ;
      L     "MAL1S024Par".Ilo.Code_ILO_Funktion0;
      L     500;
      <>I   ;
      )     ;
      SPB   F05b;
      L     "MAL1S024Par".Ilo.SetpointInt01[1];
      T     "MAL1S024Par".Par.ParIntProcess.Speed_ILO_Fan;
F05b: NOP   0;
//BRT070310 - Sollwert Frischluftklappen!
      UN    "G251M".Gr.InManual; // FRESH AIR LOUVER GERM 8
      O(    ;
      L     "MAL1S024Par".Ilo.Code_ILO_Funktion0;
      L     500;
      <>I   ;
      )     ;
      SPB   F05c;
      L     "MAL1S024Par".Ilo.SetpointInt03[1];
      T     "MAL1S024Par".Par.ParIntProcess.TarPos_ILO_FreshAir;
F05c: NOP   0;

IO5:  NOP   0;
      NOP   0;
// --- FCM 06 - Fresh air flap ---
      L     "MAL1S024Par".Ilo.ILOMode;
      L     6;
      <>I   ;
      SPB   IO6;
// man on
      U     "MAL1S024Par".Ilo.GrCMDManOn[1];
      S     "G251M".Gr.InManual; // FRESH AIR LOUVER  GERM 8
//      R     DB909.DBX 3032.0
// man off
      U     "MAL1S024Par".Ilo.GrCMDManOff[1];
      S     "G251M".Gr.CmdManualOff; // FRESH AIR LOUVER  GERM 8
      R     "G251M".Gr.InManual; // FRESH AIR LOUVER  GERM 8
      R     "G251M".USW14; // ILO-cmd
      R     "G251M".USW15; // ILO-cmd
      R     "MAL1S024Par".Ilo.GrCMDManOff[1];
      R     "MAL1S024Par".Ilo.GrCMDManAdditional.Cmd1[1];
      R     "MAL1S024Par".Ilo.GrCMDManAdditional.Cmd2[1];
// man start
      U     "MAL1S024Par".Ilo.GrCMDManStart[1];
      S     "G251M".Gr.CmdOn; // FRESH AIR LOUVER  GERM 8
      S     "G251M".Gr.CmdContinue; // FRESH AIR LOUVER  GERM 8
      R     "MAL1S024Par".Ilo.GrCMDManStart[1];
      U     "MAL1S024Par".Ilo.GrCMDManStart[2];
      R     "MAL1S024Par".Ilo.GrCMDManStart[2];

      U     "MAL1S024Par".Ilo.GrCMDManOn[1];
      R     "MAL1S024Par".Ilo.GrCMDManOn[1];
// man stop
      U     "MAL1S024Par".Ilo.GrCMDManStop[1];
      S     "G251M".Gr.CmdOff; // FRESH AIR LOUVER  GERM 8
      R     "MAL1S024Par".Ilo.GrCMDManStop[1];
// man fault reset
//BRT070310      U     "MAL1S024Par".Ilo.GrCMDManOn[17]
      U     "MAL1S024Par".Ilo.GrCMDManFaultReset[1]; //BRT070310
      S     "G251M".Gr.CmdFaultReset; // FRESH AIR LOUVER  GERM 8
      R     "MAL1S024Par".Ilo.GrCMDManFaultReset[1]; //BRT070310
// moving direction

// target position
      UN    "G251M".Gr.InManual; // FRESH AIR LOUVER  GERM 8
      SPB   F06b;
      L     "MAL1S024Par".Ilo.SetpointInt01[1];
      T     "MAL1S024Par".Par.ParIntProcess.TarPos_ILO_FreshAir;
F06b: NOP   0;

IO6:  NOP   0;
      NOP   0;
// --- FCM 09 - Floor drives ---
      L     "MAL1S024Par".Ilo.ILOMode;
      L     9;
      <>I   ;
      SPB   IO9;
// man on
      U     "MAL1S024Par".Ilo.GrCMDManOn[1];
      S     "G014G".Gr.InManual; // GENERAL ELEMENTS GERM 8
      S     "G245M".Gr.InManual; // TRAVELLING DRIVE  GERM 8
      S     "G249M".Gr.InManual; // TURNING SCREWS  GERM 8
      R     "MAL1S024Par".Ilo.GrCMDManOn[1];
// man off
      U     "MAL1S024Par".Ilo.GrCMDManOff[1];
//====>BRT070310
      S     "G014G".Gr.CmdManualOff; // GENERAL ELEMENTS GERM 8
      R     "G014G".Gr.InManual; // GENERAL ELEMENTS GERM 8
      S     "G245M".Gr.CmdManualOff; // TRAVELLING DRIVE  GERM 8
      R     "G245M".Gr.InManual; // TRAVELLING DRIVE  GERM 8
      R     "G245M".USW14; // ILO-cmd
      R     "G245M".USW15; // ILO-cmd
      S     "G249M".Gr.CmdManualOff; // TURNING SCREWS  GERM 8
      R     "G249M".Gr.InManual; // TURNING SCREWS  GERM 8
      R     "G249M".USW14; // ILO-cmd
      R     "G249M".USW15; // ILO-cmd
      R     "MAL1S024Par".Ilo.GrCMDManOff[1];
      R     "MAL1S024Par".Ilo.GrCMDManAdditional.Cmd1[1];
      R     "MAL1S024Par".Ilo.GrCMDManAdditional.Cmd2[1];
// man start
      U     "MAL1S024Par".Ilo.GrCMDManStart[1];
      S     "G014G".Gr.CmdOn; // GENERAL ELEMENTS GERM 8
      S     "G014G".Gr.CmdContinue; // GENERAL ELEMENTS GERM 8
      S     "G245M".Gr.CmdOn; // TRAVELLING DRIVE  GERM 8
      S     "G245M".Gr.CmdContinue; // TRAVELLING DRIVE  GERM 8
      S     "G249M".Gr.CmdOn; // TURNING SCREWS  GERM 8
      S     "G249M".Gr.CmdContinue; // TURNING SCREWS  GERM 8
      U     "MAL1S024Par".Ilo.GrCMDManStart[1];
      R     "MAL1S024Par".Ilo.GrCMDManStart[1];
      U     "MAL1S024Par".Ilo.GrCMDManStart[2];
      R     "MAL1S024Par".Ilo.GrCMDManStart[2];
// man stop
      U     "MAL1S024Par".Ilo.GrCMDManStop[1];
//====>BRT070310 - vom Man Off rauskopiert nach Man Stop
      O(    ;
      U(    ;
      U     "G245M".A_2811_BZS46.StTrue; // stop discharge side
      O     "G245M".A_2811_BZS46.InpTrue;
      U     "G245M".Gr.InManual;
      U     "G245M".USW14; // ILO-cmd run fwd
      )     ;
      O(    ;
      U     "G245M".A_2811_BZS44.StTrue; // stop fan side
      O     "G245M".A_2811_BZS44.InpTrue; // stop fan side
      U     "G245M".Gr.InManual;
      U     "G245M".USW15; // ILO-cmd run rev
      )     ;
      U(    ;
      L     "MAL1S024Par".Ilo.ILOMode;
//BRT070310      L     8
      L     9; //BRT070310
      ==I   ;
      )     ;
      )     ;
//<====BRT070310
      S     "G245M".Gr.CmdOff; // TRAVELLING DRIVE  GERM 8
//BRT120310      S     "G249M".Gr.CmdOff           // TURNING SCREWS  GERM 8
      R     "G245M".USW14; // ILO-cmd run fwd  //BRT120310
      R     "G245M".USW15; // ILO-cmd run rev  //BRT120310
      R     "MAL1S024Par".Ilo.GrCMDManStop[1];
// man fault reset
      U     "MAL1S024Par".Ilo.GrCMDManFaultReset[1];
      S     "G014G".Gr.CmdFaultReset; // GENERAL ELEMENTS GERM 8
      S     "G245M".Gr.CmdFaultReset; // TRAVELLING DRIVE  GERM 8
      S     "G249M".Gr.CmdFaultReset; // TURNING SCREWS  GERM 8
      R     "MAL1S024Par".Ilo.GrCMDManFaultReset[1];
// manual direction
      UN    "G245M".Gr.InManual; // TRAVELLING DRIVE  GERM 8
      SPB   f092;
      U     "MAL1S024Par".Ilo.GrCMDManAdditional.Cmd1[1];
      =     "G245M".USW14; // ILO-cmd run fwd
      U     "MAL1S024Par".Ilo.GrCMDManAdditional.Cmd2[1];
      =     "G245M".USW15; // ILO-cmd run rev
// target position
      L     "MAL1S024Par".Ilo.SetpointInt01[1];
      T     "MAL1S024Par".Par.ParIntProcess.Speed_ILO_FloorRotating;
f092: NOP   0;


IO9:  NOP   0;
// --- FCM 10 - local operating on operating panels ---
      L     "MAL1S024Par".Ilo.ILOMode;
      L     10;
      <>I   ;
      SPB   I10;
// man on
      U     "MAL1S024Par".Ilo.GrCMDManOn[1];
      S     "G014G".Gr.InManual; // GENERAL ELEMENTS GERM 8
      S     "G245M".Gr.InManual; // Traveling  Drive Germatingbox 8
      S     "G249M".Gr.InManual; // Turning Screws Germinationbox 8
      S     "G244M".Gr.InManual; // Wall locking Germatingbox 8
      S     "G242M".Gr.InManual; // Backwall moving Germatingbox 8
      S     "G243M".Gr.InManual; // Discharger locking Germatingbox 8
      R     "MAL1S024Par".Ilo.GrCMDManOn[1];
// man off
      U     "MAL1S024Par".Ilo.GrCMDManOff[1];
      S     "G014G".Gr.CmdManualOff; // GENERAL ELEMENTS GERM 8
      R     "G014G".Gr.InManual; // GENERAL ELEMENTS GERM 8
      S     "G245M".Gr.CmdManualOff; // Traveling  Drive Germatingbox 8
      R     "G245M".Gr.InManual; // Traveling  Drive Germatingbox 8
      R     "G245M".USW14; // ILO-cmd
      R     "G245M".USW15; // ILO-cmd
      S     "G249M".Gr.CmdManualOff; // Turning Screws Germinationbox 8
      R     "G249M".Gr.InManual; // Turning Screws Germinationbox 8
      R     "G249M".USW14; // ILO-cmd
      R     "G249M".USW15; // ILO-cmd
      S     "G244M".Gr.CmdManualOff; // Wall locking Germatingbox 8
      R     "G244M".Gr.InManual; // Wall locking Germatingbox 8
      S     "G243M".Gr.CmdManualOff; // Discharger locking Germatingbox 8
      R     "G243M".Gr.InManual; // Discharger locking Germatingbox 8
      S     "G242M".Gr.CmdManualOff; // Backwall moving Germatingbox 8
      R     "G242M".Gr.InManual; // Backwall moving Germatingbox 8
      R     "MAL1S024Par".Ilo.GrCMDManOff[1];
      R     "MAL1S024Par".Ilo.GrCMDManAdditional.Cmd1[1];
      R     "MAL1S024Par".Ilo.GrCMDManAdditional.Cmd2[1];
// man start
      U     "G247M".A_2811_KCL01I1.InpTrue; // pushbutton "start screws"
      S     "G014G".Gr.CmdOn; // GENERAL ELEMENTS GERM 8
      S     "G014G".Gr.CmdContinue; // GENERAL ELEMENTS GERM 8
      S     "G249M".Gr.CmdOn; // Turning Screws Germinationbox 8
      S     "G249M".Gr.CmdContinue; // Turning Screws Germinationbox 8
      S     "G245M".Gr.CmdOn; // Traveling  Drive Germatingbox 8
      S     "G245M".Gr.CmdContinue; // Traveling  Drive Germatingbox 8
      U     "MAL1S024Par".Ilo.GrCMDManStart[1];
      R     "MAL1S024Par".Ilo.GrCMDManStart[1];
      U     "MAL1S024Par".Ilo.GrCMDManStart[2];
      R     "MAL1S024Par".Ilo.GrCMDManStart[2];
// man stop
      UN    "G247M".A_2811_KCL01I2.InpTrue; // pushbutton "stop screws"  //dyk 081025 Inverted
      S     "G249M".Gr.CmdOff; // Turning Screws Germinationbox 8
      U     "MAL1S024Par".Ilo.GrCMDManStop[1];
      O(    ;
      UN    "G247M".A_2811_KCL01I3.InpTrue; // pushbutton "drive fwd"
      UN    "G247M".A_2811_KCL01I4.InpTrue; // pushbutton "drive rev"
      )     ;
      S     "G245M".Gr.CmdOff; // Traveling  Drive Germatingbox 8

      UN    "G244M".Gr.InManual; // Wall locking Germatingbox 8
      O(    ;
      UN    "G247M".A_2815_KCL01I5.InpTrue; // pushbutton "locking"
      UN    "G247M".A_2815_KCL01I6.InpTrue; // pushbutton "unlocking"
      )     ;
      S     "G244M".Gr.CmdOff; // Wall locking/unlocking Germatingbox 8

      UN    "G243M".Gr.InManual; // discharger coupling Germatingbox 8
      O(    ;
      UN    "G247M".A_2815_KCL01I4.InpTrue; // pushbutton "discharger coupling"
      UN    "G247M".A_2815_KCL01I3.InpTrue; // pushbutton "discharger uncoupling"
      )     ;
      S     "G243M".Gr.CmdOff; // discharger coupling Germatingbox 8

      UN    "G242M".Gr.InManual; // Backwall moving Germatingbox 8
      O(    ;
      UN    "G247M".A_2815_KCL01I1.InpTrue; // pushbutton "backwall lifting"
      UN    "G247M".A_2815_KCL01I2.InpTrue; // pushbutton "backwall lowerring"
      )     ;
      S     "G242M".Gr.CmdOff; // Backwall moving Germatingbox 8

      U     "MAL1S024Par".Ilo.GrCMDManStop[1];
      R     "MAL1S024Par".Ilo.GrCMDManStop[1];
// man fault reset
      U     "MAL1S024Par".Ilo.GrCMDManFaultReset[1];
      S     "G014G".Gr.CmdFaultReset; // GENERAL ELEMENTS GERM 8
      S     "G245M".Gr.CmdFaultReset; // Traveling  Drive Germatingbox 8
      S     "G249M".Gr.CmdFaultReset; // Turning Screws Germinationbox 8
      R     "MAL1S024Par".Ilo.GrCMDManFaultReset[1];
      NOP   0;
// Manual wall locking
      UN    "G244M".Gr.InManual; // Wall locking Germatingbox 8
      ON    "G247M".A_2815_KCL01I5.InpTrue; // pushbutton "locking"
      SPB   f102;
      S     "G244M".Gr.CmdOn; // Wall locking/unlocking Germatingbox 8
f102: NOP   0;
// Manual wall unlocking
      UN    "G244M".Gr.InManual; // Wall locking Germatingbox 8
      ON    "G247M".A_2815_KCL01I6.InpTrue; // pushbutton "unlocking"
      SPB   f103;
      S     "G244M".Gr.CmdOn; // Wall locking/unlocking Germatingbox 8
f103: NOP   0;
// Manual discharger coupling
      UN    "G243M".Gr.InManual; // discharger coupling Germatingbox 8
      ON    "G247M".A_2815_KCL01I4.InpTrue; // pushbutton "discharger coupling"
      SPB   f104;
      S     "G243M".Gr.CmdOn; // discharger coupling Germatingbox 8
f104: NOP   0;
// Manual discharger uncoupling
      UN    "G243M".Gr.InManual; // discharger coupling Germatingbox 8
      ON    "G247M".A_2815_KCL01I3.InpTrue; // pushbutton "discharger uncoupling"
      SPB   f105;
      S     "G243M".Gr.CmdOn; // discharger coupling Germatingbox 8
f105: NOP   0;
// Manual backwall moving
      UN    "G242M".Gr.InManual; // Backwall moving Germatingbox 8
      ON    "G247M".A_2815_KCL01I1.InpTrue; // pushbutton "backwall lifting"
      SPB   f106;
      S     "G242M".Gr.CmdOn; // Backwall moving Germatingbox 8
f106: NOP   0;
      UN    "G242M".Gr.InManual; // Backwall moving Germatingbox 8
      ON    "G247M".A_2815_KCL01I2.InpTrue; // pushbutton "backwall lowerring"
      SPB   f107;
      S     "G242M".Gr.CmdOn; // Backwall moving Germatingbox 8
f107: NOP   0;
// manual direction
      UN    "G245M".Gr.InManual; // Traveling  Drive Germatingbox 8
      O     ;
      UN    "G247M".A_2811_KCL01I3.InpTrue; // pushbutton "drive fwd"
      UN    "G247M".A_2811_KCL01I4.InpTrue; // pushbutton "drive rev"
      SPB   f109;
      U     "G247M".A_2811_KCL01I3.InpTrue; // pushbutton "drive fwd"
      =     "G245M".USW14; // ILO-cmd run fwd
      S     "G245M".Gr.CmdOn; // Traveling  Drive Germatingbox 8
      U     "G247M".A_2811_KCL01I4.InpTrue; // pushbutton "drive rev"
      =     "G245M".USW15; // ILO-cmd run rev
      S     "G245M".Gr.CmdOn; // Traveling  Drive Germatingbox 8

// target position
      L     "MAL1S024Par".Ilo.SetpointInt01[1];
      T     "MAL1S024Par".Par.ParIntProcess.Speed_ILO_FloorRotating;
f109: NOP   0;

